LIN {X 0,Y 473.655,Z 542.16,A -85,B 0,C 180,E1 -7089.139,E2 -7089.139} C_VEL
LIN {X 0,Y 473.783,Z 539.256,A -85,B 0,C 180,E1 -7090.503,E2 -7090.503} C_VEL
LIN {X 0,Y 473.901,Z 535.976,A -85,B 0,C 180,E1 -7091.646,E2 -7091.646} C_VEL
LIN {X 0,Y 474,Z 531.987,A -85,B 0,C 180,E1 -7092.75,E2 -7092.75} C_VEL
LIN {X 0,Y 474.226,Z 525.864,A -85,B 0,C 180,E1 -7094.079,E2 -7094.079} C_VEL
LIN {X 0,Y 474.493,Z 519.562,A -85,B 0,C 180,E1 -7095.197,E2 -7095.197} C_VEL
LIN {X 0,Y 474.846,Z 511.99,A -85,B 0,C 180,E1 -7096.302,E2 -7096.302} C_VEL
LIN {X 0,Y 475.225,Z 503.778,A -85,B 0,C 180,E1 -7097.296,E2 -7097.296} C_VEL
LIN {X 0,Y 475.641,Z 495.123,A -85,B 0,C 180,E1 -7098.17,E2 -7098.17} C_VEL
LIN {X 0,Y 476.009,Z 486.024,A -85,B 0,C 180,E1 -7098.934,E2 -7098.934} C_VEL
LIN {X 0,Y 476.406,Z 476.552,A -85,B 0,C 180,E1 -7099.589,E2 -7099.589} C_VEL
LIN {X 0,Y 476.754,Z 465.648,A -85,B 0,C 180,E1 -7100.186,E2 -7100.186} C_VEL
LIN {X 0,Y 477.105,Z 454.466,A -85,B 0,C 180,E1 -7100.648,E2 -7100.648} C_VEL
LIN {X 0,Y 477.363,Z 443.291,A -85,B 0,C 180,E1 -7100.975,E2 -7100.975} C_VEL
LIN {X 0,Y 477.534,Z 425.281,A -85,B 0,C 180,E1 -7101.291,E2 -7101.291} C_VEL
LIN {X 0,Y 478.031,Z 348.456,A -85,B 0,C 180,E1 -7102.453,E2 -7102.453} C_VEL
LIN {X 0,Y 475.663,Z 335.476,A -85,B 0,C 180,E1 -7102.743,E2 -7102.743} C_VEL
LIN {X 0,Y 475.427,Z 333.673,A -85,B 0,C 180,E1 -7102.844,E2 -7102.844} C_VEL
LIN {X 0,Y 476.024,Z 317.906,A -85,B 0,C 180,E1 -7105.979,E2 -7105.979} C_VEL
LIN {X 0,Y 476.244,Z 312.656,A -85,B 0,C 180,E1 -7107.039,E2 -7107.039} C_VEL
LIN {X 0,Y 474.843,Z 303.952,A -85,B 0,C 180,E1 -7108.94,E2 -7108.94} C_VEL
LIN {X 0,Y 474.859,Z 303.836,A -85,B 0,C 180,E1 -7110.848,E2 -7110.848} C_VEL
LIN {X 0,Y 474.895,Z 303.831,A -85,B 0,C 180,E1 -7112.545,E2 -7112.545} C_VEL
LIN {X 0,Y 474.772,Z 303.839,A -85,B 0,C 180,E1 -7115.948,E2 -7115.948} C_VEL
LIN {X 0,Y 474.714,Z 303.846,A -85,B 0,C 180,E1 -7118.514,E2 -7118.514} C_VEL
LIN {X 0,Y 474.706,Z 303.85,A -85,B 0,C 180,E1 -7121.962,E2 -7121.962} C_VEL
LIN {X 0,Y 474.702,Z 303.851,A -85,B 0,C 180,E1 -7125.456,E2 -7125.456} C_VEL
LIN {X 0,Y 474.667,Z 303.85,A -85,B 0,C 180,E1 -7129.01,E2 -7129.01} C_VEL
LIN {X 0,Y 474.59,Z 303.863,A -85,B 0,C 180,E1 -7131.729,E2 -7131.729} C_VEL
LIN {X 0,Y 474.656,Z 303.858,A -85,B 0,C 180,E1 -7134.493,E2 -7134.493} C_VEL
LIN {X 0,Y 474.683,Z 303.85,A -85,B 0,C 180,E1 -7137.334,E2 -7137.334} C_VEL
LIN {X 0,Y 474.607,Z 303.859,A -85,B 0,C 180,E1 -7140.23,E2 -7140.23} C_VEL
LIN {X 0,Y 474.645,Z 303.861,A -85,B 0,C 180,E1 -7143.22,E2 -7143.22} C_VEL
LIN {X 0,Y 474.586,Z 303.864,A -85,B 0,C 180,E1 -7146.324,E2 -7146.324} C_VEL
LIN {X 0,Y 474.629,Z 303.861,A -85,B 0,C 180,E1 -7149.648,E2 -7149.648} C_VEL
LIN {X 0,Y 474.607,Z 303.857,A -85,B 0,C 180,E1 -7152.935,E2 -7152.935} C_VEL
LIN {X 0,Y 474.605,Z 303.861,A -85,B 0,C 180,E1 -7155.894,E2 -7155.894} C_VEL
LIN {X 0,Y 474.624,Z 303.854,A -85,B 0,C 180,E1 -7159.042,E2 -7159.042} C_VEL
LIN {X 0,Y 474.611,Z 303.854,A -85,B 0,C 180,E1 -7161.704,E2 -7161.704} C_VEL
LIN {X 0,Y 474.624,Z 303.858,A -85,B 0,C 180,E1 -7164.726,E2 -7164.726} C_VEL
LIN {X 0,Y 474.637,Z 303.856,A -85,B 0,C 180,E1 -7167.788,E2 -7167.788} C_VEL
LIN {X 0,Y 474.608,Z 303.845,A -85,B 0,C 180,E1 -7170.889,E2 -7170.889} C_VEL
LIN {X 0,Y 474.616,Z 303.856,A -85,B 0,C 180,E1 -7173.626,E2 -7173.626} C_VEL
LIN {X 0,Y 474.637,Z 303.86,A -85,B 0,C 180,E1 -7176.642,E2 -7176.642} C_VEL
LIN {X 0,Y 474.655,Z 303.849,A -85,B 0,C 180,E1 -7180.089,E2 -7180.089} C_VEL
LIN {X 0,Y 474.637,Z 303.847,A -85,B 0,C 180,E1 -7182.774,E2 -7182.774} C_VEL
LIN {X 0,Y 474.643,Z 303.859,A -85,B 0,C 180,E1 -7185.421,E2 -7185.421} C_VEL
LIN {X 0,Y 474.706,Z 303.848,A -85,B 0,C 180,E1 -7188.037,E2 -7188.037} C_VEL
LIN {X 0,Y 474.698,Z 303.85,A -85,B 0,C 180,E1 -7191.486,E2 -7191.486} C_VEL
LIN {X 0,Y 474.742,Z 303.836,A -85,B 0,C 180,E1 -7194.052,E2 -7194.052} C_VEL
LIN {X 0,Y 474.876,Z 303.824,A -85,B 0,C 180,E1 -7197.455,E2 -7197.455} C_VEL
LIN {X 0,Y 474.884,Z 303.828,A -85,B 0,C 180,E1 -7200,E2 -7200} C_VEL
LIN {X 0,Y 474.874,Z 303.828,A -85,B 0,C 180,E1 -7202.544,E2 -7202.544} C_VEL
LIN {X 0,Y 474.76,Z 303.83,A -85,B 0,C 180,E1 -7205.948,E2 -7205.948} C_VEL
LIN {X 0,Y 474.703,Z 303.847,A -85,B 0,C 180,E1 -7208.514,E2 -7208.514} C_VEL
LIN {X 0,Y 474.705,Z 303.847,A -85,B 0,C 180,E1 -7211.962,E2 -7211.962} C_VEL
LIN {X 0,Y 474.681,Z 303.845,A -85,B 0,C 180,E1 -7215.456,E2 -7215.456} C_VEL
LIN {X 0,Y 474.66,Z 303.853,A -85,B 0,C 180,E1 -7219.01,E2 -7219.01} C_VEL
LIN {X 0,Y 474.588,Z 303.863,A -85,B 0,C 180,E1 -7221.729,E2 -7221.729} C_VEL
LIN {X 0,Y 474.625,Z 303.857,A -85,B 0,C 180,E1 -7224.494,E2 -7224.494} C_VEL
LIN {X 0,Y 474.598,Z 303.863,A -85,B 0,C 180,E1 -7227.326,E2 -7227.326} C_VEL
LIN {X 0,Y 474.594,Z 303.858,A -85,B 0,C 180,E1 -7230.231,E2 -7230.231} C_VEL
LIN {X 0,Y 474.614,Z 303.864,A -85,B 0,C 180,E1 -7233.222,E2 -7233.222} C_VEL
LIN {X 0,Y 474.58,Z 303.861,A -85,B 0,C 180,E1 -7236.324,E2 -7236.324} C_VEL
LIN {X 0,Y 474.6,Z 303.866,A -85,B 0,C 180,E1 -7239.643,E2 -7239.643} C_VEL
LIN {X 0,Y 474.574,Z 303.868,A -85,B 0,C 180,E1 -7242.23,E2 -7242.23} C_VEL
LIN {X 0,Y 474.611,Z 303.859,A -85,B 0,C 180,E1 -7245.298,E2 -7245.298} C_VEL
LIN {X 0,Y 474.589,Z 303.866,A -85,B 0,C 180,E1 -7248.211,E2 -7248.211} C_VEL
LIN {X 0,Y 474.6,Z 303.862,A -85,B 0,C 180,E1 -7251.541,E2 -7251.541} C_VEL
LIN {X 0,Y 474.617,Z 303.862,A -85,B 0,C 180,E1 -7254.725,E2 -7254.725} C_VEL
LIN {X 0,Y 474.625,Z 303.864,A -85,B 0,C 180,E1 -7257.787,E2 -7257.787} C_VEL
LIN {X 0,Y 474.604,Z 303.864,A -85,B 0,C 180,E1 -7260.888,E2 -7260.888} C_VEL
LIN {X 0,Y 474.588,Z 303.868,A -85,B 0,C 180,E1 -7263.624,E2 -7263.624} C_VEL
LIN {X 0,Y 474.659,Z 304.014,A -85,B 0,C 180,E1 -7265.274,E2 -7265.274} C_VEL
LIN {X 0,Y 476.452,Z 313.581,A -85,B 0,C 180,E1 -7267.219,E2 -7267.219} C_VEL
LIN {X 0,Y 476.572,Z 317.444,A -85,B 0,C 180,E1 -7267.956,E2 -7267.956} C_VEL
LIN {X 0,Y 475.739,Z 335.291,A -85,B 0,C 180,E1 -7271.258,E2 -7271.258} C_VEL
LIN {X 0,Y 475.396,Z 346.264,A -85,B 0,C 180,E1 -7273.226,E2 -7273.226} C_VEL
LIN {X 0,Y 476.707,Z 354.719,A -85,B 0,C 180,E1 -7273.437,E2 -7273.437} C_VEL
LIN {X 0,Y 478.041,Z 363.134,A -85,B 0,C 180,E1 -7273.613,E2 -7273.613} C_VEL
LIN {X 0,Y 477.426,Z 452.372,A -85,B 0,C 180,E1 -7274.99,E2 -7274.99} C_VEL
LIN {X 0,Y 477.205,Z 462.229,A -85,B 0,C 180,E1 -7275.228,E2 -7275.228} C_VEL
LIN {X 0,Y 476.875,Z 472.814,A -85,B 0,C 180,E1 -7275.599,E2 -7275.599} C_VEL
LIN {X 0,Y 476.578,Z 482.083,A -85,B 0,C 180,E1 -7276.026,E2 -7276.026} C_VEL
LIN {X 0,Y 476.14,Z 493.305,A -85,B 0,C 180,E1 -7276.698,E2 -7276.698} C_VEL
LIN {X 0,Y 475.741,Z 502.94,A -85,B 0,C 180,E1 -7277.417,E2 -7277.417} C_VEL
LIN {X 0,Y 475.317,Z 512.31,A -85,B 0,C 180,E1 -7278.27,E2 -7278.27} C_VEL
LIN {X 0,Y 474.979,Z 520.193,A -85,B 0,C 180,E1 -7279.126,E2 -7279.126} C_VEL
LIN {X 0,Y 474.598,Z 528.371,A -85,B 0,C 180,E1 -7280.195,E2 -7280.195} C_VEL
LIN {X 0,Y 474.314,Z 535.182,A -85,B 0,C 180,E1 -7281.264,E2 -7281.264} C_VEL
LIN {X 0,Y 474.069,Z 540.876,A -85,B 0,C 180,E1 -7282.332,E2 -7282.332} C_VEL
LIN {X 0,Y 473.929,Z 545.951,A -85,B 0,C 180,E1 -7283.49,E2 -7283.49} C_VEL
LIN {X 0,Y 473.834,Z 550.733,A -85,B 0,C 180,E1 -7284.894,E2 -7284.894} C_VEL
LIN {X 0,Y 473.733,Z 553.044,A -85,B 0,C 180,E1 -7285.746,E2 -7285.746} C_VEL
LIN {X 0,Y 473.717,Z 556.305,A -85,B 0,C 180,E1 -7287.449,E2 -7287.449} C_VEL
LIN {X 0,Y 473.681,Z 557.843,A -85,B 0,C 180,E1 -7289.15,E2 -7289.15} C_VEL
LIN {X 0,Y 473.664,Z 558.137,A -85,B 0,C 180,E1 -7290,E2 -7290} C_VEL
LIN {X 0,Y 473.687,Z 557.271,A -85,B 0,C 180,E1 -7291.7,E2 -7291.7} C_VEL
LIN {X 0,Y 473.717,Z 556.304,A -85,B 0,C 180,E1 -7292.551,E2 -7292.551} C_VEL
LIN {X 0,Y 473.733,Z 553.044,A -85,B 0,C 180,E1 -7294.254,E2 -7294.254} C_VEL
LIN {X 0,Y 473.868,Z 549.438,A -85,B 0,C 180,E1 -7295.532,E2 -7295.532} C_VEL
LIN {X 0,Y 473.972,Z 544.709,A -85,B 0,C 180,E1 -7296.813,E2 -7296.813} C_VEL
LIN {X 0,Y 474.17,Z 538.712,A -85,B 0,C 180,E1 -7298.094,E2 -7298.094} C_VEL
LIN {X 0,Y 474.4,Z 532.643,A -85,B 0,C 180,E1 -7299.164,E2 -7299.164} C_VEL
LIN {X 0,Y 474.715,Z 525.324,A -85,B 0,C 180,E1 -7300.233,E2 -7300.233} C_VEL
LIN {X 0,Y 475.171,Z 516.421,A -85,B 0,C 180,E1 -7301.302,E2 -7301.302} C_VEL
LIN {X 0,Y 475.602,Z 507.884,A -85,B 0,C 180,E1 -7302.155,E2 -7302.155} C_VEL
LIN {X 0,Y 475.929,Z 498.455,A -85,B 0,C 180,E1 -7302.939,E2 -7302.939} C_VEL
LIN {X 0,Y 476.278,Z 489.644,A -85,B 0,C 180,E1 -7303.547,E2 -7303.547} C_VEL
LIN {X 0,Y 476.732,Z 477.751,A -85,B 0,C 180,E1 -7304.187,E2 -7304.187} C_VEL
LIN {X 0,Y 477.051,Z 467.383,A -85,B 0,C 180,E1 -7304.613,E2 -7304.613} C_VEL
LIN {X 0,Y 477.397,Z 456.571,A -85,B 0,C 180,E1 -7304.929,E2 -7304.929} C_VEL
LIN {X 0,Y 477.55,Z 438.378,A -85,B 0,C 180,E1 -7305.252,E2 -7305.252} C_VEL
LIN {X 0,Y 477.994,Z 362.184,A -85,B 0,C 180,E1 -7306.417,E2 -7306.417} C_VEL
LIN {X 0,Y 475.357,Z 346.208,A -85,B 0,C 180,E1 -7306.791,E2 -7306.791} C_VEL
LIN {X 0,Y 475.635,Z 337.488,A -85,B 0,C 180,E1 -7308.3,E2 -7308.3} C_VEL
LIN {X 0,Y 476.378,Z 319.034,A -85,B 0,C 180,E1 -7311.653,E2 -7311.653} C_VEL
LIN {X 0,Y 476.369,Z 312.947,A -85,B 0,C 180,E1 -7312.785,E2 -7312.785} C_VEL
LIN {X 0,Y 474.654,Z 303.952,A -85,B 0,C 180,E1 -7314.61,E2 -7314.61} C_VEL
LIN {X 0,Y 474.634,Z 303.862,A -85,B 0,C 180,E1 -7317.324,E2 -7317.324} C_VEL
LIN {X 0,Y 474.599,Z 303.869,A -85,B 0,C 180,E1 -7320.231,E2 -7320.231} C_VEL
LIN {X 0,Y 474.622,Z 303.86,A -85,B 0,C 180,E1 -7323.222,E2 -7323.222} C_VEL
LIN {X 0,Y 474.586,Z 303.869,A -85,B 0,C 180,E1 -7326.324,E2 -7326.324} C_VEL
LIN {X 0,Y 474.611,Z 303.857,A -85,B 0,C 180,E1 -7329.646,E2 -7329.646} C_VEL
LIN {X 0,Y 474.598,Z 303.863,A -85,B 0,C 180,E1 -7332.234,E2 -7332.234} C_VEL
LIN {X 0,Y 474.62,Z 303.867,A -85,B 0,C 180,E1 -7335.297,E2 -7335.297} C_VEL
LIN {X 0,Y 474.619,Z 303.858,A -85,B 0,C 180,E1 -7338.215,E2 -7338.215} C_VEL
LIN {X 0,Y 474.611,Z 303.866,A -85,B 0,C 180,E1 -7341.543,E2 -7341.543} C_VEL
LIN {X 0,Y 474.628,Z 303.856,A -85,B 0,C 180,E1 -7344.726,E2 -7344.726} C_VEL
LIN {X 0,Y 474.635,Z 303.86,A -85,B 0,C 180,E1 -7347.788,E2 -7347.788} C_VEL
LIN {X 0,Y 474.624,Z 303.861,A -85,B 0,C 180,E1 -7350.885,E2 -7350.885} C_VEL
LIN {X 0,Y 474.66,Z 303.853,A -85,B 0,C 180,E1 -7353.629,E2 -7353.629} C_VEL
LIN {X 0,Y 474.635,Z 303.862,A -85,B 0,C 180,E1 -7356.642,E2 -7356.642} C_VEL
LIN {X 0,Y 474.658,Z 303.853,A -85,B 0,C 180,E1 -7360.09,E2 -7360.09} C_VEL
LIN {X 0,Y 474.652,Z 303.854,A -85,B 0,C 180,E1 -7362.775,E2 -7362.775} C_VEL
LIN {X 0,Y 474.654,Z 303.86,A -85,B 0,C 180,E1 -7365.421,E2 -7365.421} C_VEL
LIN {X 0,Y 474.706,Z 303.853,A -85,B 0,C 180,E1 -7368.038,E2 -7368.038} C_VEL
LIN {X 0,Y 474.73,Z 303.843,A -85,B 0,C 180,E1 -7371.487,E2 -7371.487} C_VEL
LIN {X 0,Y 474.781,Z 303.847,A -85,B 0,C 180,E1 -7374.053,E2 -7374.053} C_VEL
LIN {X 0,Y 474.896,Z 303.824,A -85,B 0,C 180,E1 -7377.456,E2 -7377.456} C_VEL
LIN {X 0,Y 474.914,Z 303.822,A -85,B 0,C 180,E1 -7380,E2 -7380} C_VEL
LIN {X 0,Y 474.896,Z 303.83,A -85,B 0,C 180,E1 -7382.545,E2 -7382.545} C_VEL
LIN {X 0,Y 474.783,Z 303.838,A -85,B 0,C 180,E1 -7385.948,E2 -7385.948} C_VEL
LIN {X 0,Y 474.73,Z 303.845,A -85,B 0,C 180,E1 -7388.514,E2 -7388.514} C_VEL
LIN {X 0,Y 474.706,Z 303.848,A -85,B 0,C 180,E1 -7391.963,E2 -7391.963} C_VEL
LIN {X 0,Y 474.702,Z 303.855,A -85,B 0,C 180,E1 -7395.456,E2 -7395.456} C_VEL
LIN {X 0,Y 474.667,Z 303.852,A -85,B 0,C 180,E1 -7399.01,E2 -7399.01} C_VEL
LIN {X 0,Y 474.59,Z 303.867,A -85,B 0,C 180,E1 -7401.729,E2 -7401.729} C_VEL
LIN {X 0,Y 474.642,Z 303.863,A -85,B 0,C 180,E1 -7404.494,E2 -7404.494} C_VEL
LIN {X 0,Y 474.656,Z 303.849,A -85,B 0,C 180,E1 -7407.328,E2 -7407.328} C_VEL
LIN {X 0,Y 474.606,Z 303.865,A -85,B 0,C 180,E1 -7410.81,E2 -7410.81} C_VEL
LIN {X 0,Y 474.626,Z 303.862,A -85,B 0,C 180,E1 -7413.222,E2 -7413.222} C_VEL
LIN {X 0,Y 474.589,Z 303.863,A -85,B 0,C 180,E1 -7416.324,E2 -7416.324} C_VEL
LIN {X 0,Y 474.628,Z 303.865,A -85,B 0,C 180,E1 -7419.648,E2 -7419.648} C_VEL
LIN {X 0,Y 474.635,Z 303.864,A -85,B 0,C 180,E1 -7422.932,E2 -7422.932} C_VEL
LIN {X 0,Y 474.659,Z 304.019,A -85,B 0,C 180,E1 -7423.755,E2 -7423.755} C_VEL
LIN {X 0,Y 475.868,Z 310.991,A -85,B 0,C 180,E1 -7425.146,E2 -7425.146} C_VEL
LIN {X 0,Y 475.559,Z 326.316,A -85,B 0,C 180,E1 -7427.972,E2 -7427.972} C_VEL
LIN {X 0,Y 475.397,Z 333.585,A -85,B 0,C 180,E1 -7429.262,E2 -7429.262} C_VEL
LIN {X 0,Y 478.15,Z 348.867,A -85,B 0,C 180,E1 -7429.624,E2 -7429.624} C_VEL
LIN {X 0,Y 477.411,Z 440.006,A -85,B 0,C 180,E1 -7431.037,E2 -7431.037} C_VEL
LIN {X 0,Y 477.184,Z 449.685,A -85,B 0,C 180,E1 -7431.277,E2 -7431.277} C_VEL
LIN {X 0,Y 477.012,Z 458.923,A -85,B 0,C 180,E1 -7431.598,E2 -7431.598} C_VEL
LIN {X 0,Y 476.643,Z 470.39,A -85,B 0,C 180,E1 -7432.139,E2 -7432.139} C_VEL
LIN {X 0,Y 476.508,Z 473.811,A -85,B 0,C 180,E1 -7432.334,E2 -7432.334} C_VEL
LIN {X 0,Y 475.642,Z 479.172,A -85,B 0,C 180,E1 -7432.636,E2 -7432.636} C_VEL
LIN {X 0,Y 472.465,Z 487.502,A -85,B 0,C 180,E1 -7433.15,E2 -7433.15} C_VEL
LIN {X 0,Y 469.282,Z 495.478,A -85,B 0,C 180,E1 -7433.757,E2 -7433.757} C_VEL
LIN {X 0,Y 468.416,Z 500.019,A -85,B 0,C 180,E1 -7434.2,E2 -7434.2} C_VEL
LIN {X 0,Y 468.094,Z 506.843,A -85,B 0,C 180,E1 -7434.95,E2 -7434.95} C_VEL
LIN {X 0,Y 467.706,Z 514.606,A -85,B 0,C 180,E1 -7435.967,E2 -7435.967} C_VEL
LIN {X 0,Y 467.348,Z 522.436,A -85,B 0,C 180,E1 -7437.223,E2 -7437.223} C_VEL
LIN {X 0,Y 467.109,Z 527.684,A -85,B 0,C 180,E1 -7438.224,E2 -7438.224} C_VEL
LIN {X 0,Y 466.952,Z 532.064,A -85,B 0,C 180,E1 -7439.221,E2 -7439.221} C_VEL
LIN {X 0,Y 466.75,Z 537.603,A -85,B 0,C 180,E1 -7440.847,E2 -7440.847} C_VEL
LIN {X 0,Y 466.651,Z 540.911,A -85,B 0,C 180,E1 -7442.168,E2 -7442.168} C_VEL
LIN {X 0,Y 466.561,Z 542.715,A -85,B 0,C 180,E1 -7443.134,E2 -7443.134} C_VEL
LIN {X 0,Y 466.466,Z 544.498,A -85,B 0,C 180,E1 -7444.688,E2 -7444.688} C_VEL
LIN {X 0,Y 466.46,Z 544.981,A -85,B 0,C 180,E1 -7445.996,E2 -7445.996} C_VEL
LIN {X 0,Y 466.474,Z 544,A -85,B 0,C 180,E1 -7447.873,E2 -7447.873} C_VEL
LIN {X 0,Y 466.548,Z 542.49,A -85,B 0,C 180,E1 -7449.06,E2 -7449.06} C_VEL
LIN {X 0,Y 466.657,Z 540.335,A -85,B 0,C 180,E1 -7450.193,E2 -7450.193} C_VEL
LIN {X 0,Y 466.818,Z 536.626,A -85,B 0,C 180,E1 -7451.569,E2 -7451.569} C_VEL
LIN {X 0,Y 467.011,Z 530.719,A -85,B 0,C 180,E1 -7453.161,E2 -7453.161} C_VEL
LIN {X 0,Y 467.252,Z 524.78,A -85,B 0,C 180,E1 -7454.417,E2 -7454.417} C_VEL
LIN {X 0,Y 467.492,Z 519.119,A -85,B 0,C 180,E1 -7455.415,E2 -7455.415} C_VEL
LIN {X 0,Y 467.858,Z 511.447,A -85,B 0,C 180,E1 -7456.536,E2 -7456.536} C_VEL
LIN {X 0,Y 468.244,Z 503.727,A -85,B 0,C 180,E1 -7457.479,E2 -7457.479} C_VEL
LIN {X 0,Y 468.713,Z 494.292,A -85,B 0,C 180,E1 -7458.431,E2 -7458.431} C_VEL
LIN {X 0,Y 469.134,Z 484.967,A -85,B 0,C 180,E1 -7459.207,E2 -7459.207} C_VEL
LIN {X 0,Y 469.537,Z 475.223,A -85,B 0,C 180,E1 -7459.871,E2 -7459.871} C_VEL
LIN {X 0,Y 469.891,Z 465.105,A -85,B 0,C 180,E1 -7460.422,E2 -7460.422} C_VEL
LIN {X 0,Y 470.226,Z 454.023,A -85,B 0,C 180,E1 -7460.88,E2 -7460.88} C_VEL
LIN {X 0,Y 470.517,Z 443.081,A -85,B 0,C 180,E1 -7461.199,E2 -7461.199} C_VEL
LIN {X 0,Y 470.709,Z 424.841,A -85,B 0,C 180,E1 -7461.521,E2 -7461.521} C_VEL
LIN {X 0,Y 471.238,Z 349.532,A -85,B 0,C 180,E1 -7462.677,E2 -7462.677} C_VEL
LIN {X 0,Y 468.66,Z 335.347,A -85,B 0,C 180,E1 -7463.002,E2 -7463.002} C_VEL
LIN {X 0,Y 468.457,Z 333.704,A -85,B 0,C 180,E1 -7463.107,E2 -7463.107} C_VEL
LIN {X 0,Y 469.279,Z 315.538,A -85,B 0,C 180,E1 -7466.781,E2 -7466.781} C_VEL
LIN {X 0,Y 468.819,Z 310.492,A -85,B 0,C 180,E1 -7467.852,E2 -7467.852} C_VEL
LIN {X 0,Y 467.806,Z 304.81,A -85,B 0,C 180,E1 -7469.139,E2 -7469.139} C_VEL
LIN {X 0,Y 467.811,Z 304.714,A -85,B 0,C 180,E1 -7470.861,E2 -7470.861} C_VEL
LIN {X 0,Y 467.861,Z 304.707,A -85,B 0,C 180,E1 -7472.583,E2 -7472.583} C_VEL
LIN {X 0,Y 467.736,Z 304.715,A -85,B 0,C 180,E1 -7476.038,E2 -7476.038} C_VEL
LIN {X 0,Y 467.672,Z 304.724,A -85,B 0,C 180,E1 -7478.643,E2 -7478.643} C_VEL
LIN {X 0,Y 467.658,Z 304.726,A -85,B 0,C 180,E1 -7482.146,E2 -7482.146} C_VEL
LIN {X 0,Y 467.641,Z 304.733,A -85,B 0,C 180,E1 -7485.695,E2 -7485.695} C_VEL
LIN {X 0,Y 467.619,Z 304.729,A -85,B 0,C 180,E1 -7488.765,E2 -7488.765} C_VEL
LIN {X 0,Y 467.582,Z 304.736,A -85,B 0,C 180,E1 -7491.268,E2 -7491.268} C_VEL
LIN {X 0,Y 467.572,Z 304.734,A -85,B 0,C 180,E1 -7493.943,E2 -7493.943} C_VEL
LIN {X 0,Y 467.618,Z 304.738,A -85,B 0,C 180,E1 -7496.8,E2 -7496.8} C_VEL
LIN {X 0,Y 467.556,Z 304.739,A -85,B 0,C 180,E1 -7499.738,E2 -7499.738} C_VEL
LIN {X 0,Y 467.585,Z 304.735,A -85,B 0,C 180,E1 -7502.758,E2 -7502.758} C_VEL
LIN {X 0,Y 467.552,Z 304.745,A -85,B 0,C 180,E1 -7505.89,E2 -7505.89} C_VEL
LIN {X 0,Y 467.583,Z 304.735,A -85,B 0,C 180,E1 -7509.145,E2 -7509.145} C_VEL
LIN {X 0,Y 467.588,Z 304.735,A -85,B 0,C 180,E1 -7512.567,E2 -7512.567} C_VEL
LIN {X 0,Y 467.567,Z 304.739,A -85,B 0,C 180,E1 -7515.053,E2 -7515.053} C_VEL
LIN {X 0,Y 467.575,Z 304.74,A -85,B 0,C 180,E1 -7518.597,E2 -7518.597} C_VEL
LIN {X 0,Y 467.566,Z 304.73,A -85,B 0,C 180,E1 -7521.955,E2 -7521.955} C_VEL
LIN {X 0,Y 467.561,Z 304.744,A -85,B 0,C 180,E1 -7525.167,E2 -7525.167} C_VEL
LIN {X 0,Y 467.585,Z 304.729,A -85,B 0,C 180,E1 -7528.26,E2 -7528.26} C_VEL
LIN {X 0,Y 467.557,Z 304.724,A -85,B 0,C 180,E1 -7531.249,E2 -7531.249} C_VEL
LIN {X 0,Y 467.585,Z 304.74,A -85,B 0,C 180,E1 -7534.158,E2 -7534.158} C_VEL
LIN {X 0,Y 467.578,Z 304.736,A -85,B 0,C 180,E1 -7536.996,E2 -7536.996} C_VEL
LIN {X 0,Y 467.624,Z 304.723,A -85,B 0,C 180,E1 -7539.777,E2 -7539.777} C_VEL
LIN {X 0,Y 467.597,Z 304.719,A -85,B 0,C 180,E1 -7542.506,E2 -7542.506} C_VEL
LIN {X 0,Y 467.603,Z 304.737,A -85,B 0,C 180,E1 -7545.196,E2 -7545.196} C_VEL
LIN {X 0,Y 467.658,Z 304.727,A -85,B 0,C 180,E1 -7547.854,E2 -7547.854} C_VEL
LIN {X 0,Y 467.658,Z 304.726,A -85,B 0,C 180,E1 -7551.357,E2 -7551.357} C_VEL
LIN {X 0,Y 467.706,Z 304.711,A -85,B 0,C 180,E1 -7553.962,E2 -7553.962} C_VEL
LIN {X 0,Y 467.817,Z 304.703,A -85,B 0,C 180,E1 -7557.417,E2 -7557.417} C_VEL
LIN {X 0,Y 467.854,Z 304.704,A -85,B 0,C 180,E1 -7560,E2 -7560} C_VEL
LIN {X 0,Y 467.815,Z 304.706,A -85,B 0,C 180,E1 -7562.583,E2 -7562.583} C_VEL
LIN {X 0,Y 467.724,Z 304.707,A -85,B 0,C 180,E1 -7566.037,E2 -7566.037} C_VEL
LIN {X 0,Y 467.662,Z 304.725,A -85,B 0,C 180,E1 -7568.643,E2 -7568.643} C_VEL
LIN {X 0,Y 467.657,Z 304.724,A -85,B 0,C 180,E1 -7572.145,E2 -7572.145} C_VEL
LIN {X 0,Y 467.606,Z 304.727,A -85,B 0,C 180,E1 -7575.696,E2 -7575.696} C_VEL
LIN {X 0,Y 467.62,Z 304.731,A -85,B 0,C 180,E1 -7579.308,E2 -7579.308} C_VEL
LIN {X 0,Y 467.535,Z 304.745,A -85,B 0,C 180,E1 -7582.074,E2 -7582.074} C_VEL
LIN {X 0,Y 467.555,Z 304.74,A -85,B 0,C 180,E1 -7584.89,E2 -7584.89} C_VEL
LIN {X 0,Y 467.545,Z 304.74,A -85,B 0,C 180,E1 -7587.774,E2 -7587.774} C_VEL
LIN {X 0,Y 467.547,Z 304.741,A -85,B 0,C 180,E1 -7591.04,E2 -7591.04} C_VEL
LIN {X 0,Y 467.575,Z 304.737,A -85,B 0,C 180,E1 -7594.239,E2 -7594.239} C_VEL
LIN {X 0,Y 467.536,Z 304.74,A -85,B 0,C 180,E1 -7597.184,E2 -7597.184} C_VEL
LIN {X 0,Y 467.555,Z 304.743,A -85,B 0,C 180,E1 -7600.267,E2 -7600.267} C_VEL
LIN {X 0,Y 467.516,Z 304.745,A -85,B 0,C 180,E1 -7602.568,E2 -7602.568} C_VEL
LIN {X 0,Y 467.56,Z 304.739,A -85,B 0,C 180,E1 -7605.052,E2 -7605.052} C_VEL
LIN {X 0,Y 467.558,Z 304.745,A -85,B 0,C 180,E1 -7608.726,E2 -7608.726} C_VEL
LIN {X 0,Y 467.553,Z 304.739,A -85,B 0,C 180,E1 -7611.954,E2 -7611.954} C_VEL
LIN {X 0,Y 467.554,Z 304.747,A -85,B 0,C 180,E1 -7615.166,E2 -7615.166} C_VEL
LIN {X 0,Y 467.576,Z 304.738,A -85,B 0,C 180,E1 -7618.259,E2 -7618.259} C_VEL
LIN {X 0,Y 467.552,Z 304.745,A -85,B 0,C 180,E1 -7621.249,E2 -7621.249} C_VEL
LIN {X 0,Y 467.565,Z 304.745,A -85,B 0,C 180,E1 -7624.157,E2 -7624.157} C_VEL
LIN {X 0,Y 467.617,Z 304.876,A -85,B 0,C 180,E1 -7625.061,E2 -7625.061} C_VEL
LIN {X 0,Y 469.618,Z 315.892,A -85,B 0,C 180,E1 -7627.334,E2 -7627.334} C_VEL
LIN {X 0,Y 469.158,Z 326.746,A -85,B 0,C 180,E1 -7629.388,E2 -7629.388} C_VEL
LIN {X 0,Y 468.442,Z 343.624,A -85,B 0,C 180,E1 -7632.539,E2 -7632.539} C_VEL
LIN {X 0,Y 468.408,Z 346.284,A -85,B 0,C 180,E1 -7632.98,E2 -7632.98} C_VEL
LIN {X 0,Y 471.217,Z 363.856,A -85,B 0,C 180,E1 -7633.385,E2 -7633.385} C_VEL
LIN {X 0,Y 470.588,Z 452.076,A -85,B 0,C 180,E1 -7634.766,E2 -7634.766} C_VEL
LIN {X 0,Y 470.35,Z 462.005,A -85,B 0,C 180,E1 -7635.008,E2 -7635.008} C_VEL
LIN {X 0,Y 470.004,Z 472.627,A -85,B 0,C 180,E1 -7635.384,E2 -7635.384} C_VEL
LIN {X 0,Y 469.697,Z 481.92,A -85,B 0,C 180,E1 -7635.817,E2 -7635.817} C_VEL
LIN {X 0,Y 469.224,Z 493.159,A -85,B 0,C 180,E1 -7636.499,E2 -7636.499} C_VEL
LIN {X 0,Y 468.853,Z 502.059,A -85,B 0,C 180,E1 -7637.162,E2 -7637.162} C_VEL
LIN {X 0,Y 468.357,Z 512.184,A -85,B 0,C 180,E1 -7638.093,E2 -7638.093} C_VEL
LIN {X 0,Y 467.956,Z 520.072,A -85,B 0,C 180,E1 -7638.96,E2 -7638.96} C_VEL
LIN {X 0,Y 467.59,Z 528.255,A -85,B 0,C 180,E1 -7640.046,E2 -7640.046} C_VEL
LIN {X 0,Y 467.279,Z 535.069,A -85,B 0,C 180,E1 -7641.132,E2 -7641.132} C_VEL
LIN {X 0,Y 467.022,Z 540.766,A -85,B 0,C 180,E1 -7642.216,E2 -7642.216} C_VEL
LIN {X 0,Y 466.844,Z 546.236,A -85,B 0,C 180,E1 -7643.502,E2 -7643.502} C_VEL
LIN {X 0,Y 466.767,Z 550.629,A -85,B 0,C 180,E1 -7644.817,E2 -7644.817} C_VEL
LIN {X 0,Y 466.645,Z 552.94,A -85,B 0,C 180,E1 -7645.681,E2 -7645.681} C_VEL
LIN {X 0,Y 466.638,Z 556.205,A -85,B 0,C 180,E1 -7647.41,E2 -7647.41} C_VEL
LIN {X 0,Y 466.583,Z 557.743,A -85,B 0,C 180,E1 -7649.137,E2 -7649.137} C_VEL
LIN {X 0,Y 466.593,Z 558.038,A -85,B 0,C 180,E1 -7650,E2 -7650} C_VEL
LIN {X 0,Y 466.597,Z 557.173,A -85,B 0,C 180,E1 -7651.726,E2 -7651.726} C_VEL
LIN {X 0,Y 466.638,Z 556.205,A -85,B 0,C 180,E1 -7652.59,E2 -7652.59} C_VEL
LIN {X 0,Y 466.645,Z 552.945,A -85,B 0,C 180,E1 -7654.319,E2 -7654.319} C_VEL
LIN {X 0,Y 466.782,Z 549.338,A -85,B 0,C 180,E1 -7655.616,E2 -7655.616} C_VEL
LIN {X 0,Y 466.907,Z 544.609,A -85,B 0,C 180,E1 -7656.916,E2 -7656.916} C_VEL
LIN {X 0,Y 467.112,Z 538.61,A -85,B 0,C 180,E1 -7658.218,E2 -7658.218} C_VEL
LIN {X 0,Y 467.367,Z 532.54,A -85,B 0,C 180,E1 -7659.303,E2 -7659.303} C_VEL
LIN {X 0,Y 467.693,Z 525.222,A -85,B 0,C 180,E1 -7660.389,E2 -7660.389} C_VEL
LIN {X 0,Y 468.198,Z 516.324,A -85,B 0,C 180,E1 -7661.472,E2 -7661.472} C_VEL
LIN {X 0,Y 468.64,Z 508.001,A -85,B 0,C 180,E1 -7662.32,E2 -7662.32} C_VEL
LIN {X 0,Y 469.04,Z 497.629,A -85,B 0,C 180,E1 -7663.187,E2 -7663.187} C_VEL
LIN {X 0,Y 469.426,Z 487.695,A -85,B 0,C 180,E1 -7663.86,E2 -7663.86} C_VEL
LIN {X 0,Y 469.852,Z 477.695,A -85,B 0,C 180,E1 -7664.399,E2 -7664.399} C_VEL
LIN {X 0,Y 470.204,Z 466.518,A -85,B 0,C 180,E1 -7664.858,E2 -7664.858} C_VEL
LIN {X 0,Y 470.529,Z 456.577,A -85,B 0,C 180,E1 -7665.152,E2 -7665.152} C_VEL
LIN {X 0,Y 470.715,Z 438.43,A -85,B 0,C 180,E1 -7665.479,E2 -7665.479} C_VEL
LIN {X 0,Y 471.125,Z 362.415,A -85,B 0,C 180,E1 -7666.661,E2 -7666.661} C_VEL
LIN {X 0,Y 468.401,Z 346.178,A -85,B 0,C 180,E1 -7667.046,E2 -7667.046} C_VEL
LIN {X 0,Y 468.418,Z 343.519,A -85,B 0,C 180,E1 -7667.462,E2 -7667.462} C_VEL
LIN {X 0,Y 469.04,Z 328.808,A -85,B 0,C 180,E1 -7670.159,E2 -7670.159} C_VEL
LIN {X 0,Y 469.551,Z 315.308,A -85,B 0,C 180,E1 -7672.669,E2 -7672.669} C_VEL
LIN {X 0,Y 467.603,Z 304.959,A -85,B 0,C 180,E1 -7674.769,E2 -7674.769} C_VEL
LIN {X 0,Y 467.576,Z 304.744,A -85,B 0,C 180,E1 -7677.772,E2 -7677.772} C_VEL
LIN {X 0,Y 467.564,Z 304.74,A -85,B 0,C 180,E1 -7681.045,E2 -7681.045} C_VEL
LIN {X 0,Y 467.575,Z 304.74,A -85,B 0,C 180,E1 -7684.24,E2 -7684.24} C_VEL
LIN {X 0,Y 467.546,Z 304.744,A -85,B 0,C 180,E1 -7687.186,E2 -7687.186} C_VEL
LIN {X 0,Y 467.57,Z 304.735,A -85,B 0,C 180,E1 -7690.265,E2 -7690.265} C_VEL
LIN {X 0,Y 467.549,Z 304.743,A -85,B 0,C 180,E1 -7693.745,E2 -7693.745} C_VEL
LIN {X 0,Y 467.555,Z 304.739,A -85,B 0,C 180,E1 -7696.256,E2 -7696.256} C_VEL
LIN {X 0,Y 467.577,Z 304.734,A -85,B 0,C 180,E1 -7698.723,E2 -7698.723} C_VEL
LIN {X 0,Y 467.565,Z 304.745,A -85,B 0,C 180,E1 -7701.956,E2 -7701.956} C_VEL
LIN {X 0,Y 467.567,Z 304.735,A -85,B 0,C 180,E1 -7705.168,E2 -7705.168} C_VEL
LIN {X 0,Y 467.582,Z 304.74,A -85,B 0,C 180,E1 -7708.26,E2 -7708.26} C_VEL
LIN {X 0,Y 467.577,Z 304.736,A -85,B 0,C 180,E1 -7711.251,E2 -7711.251} C_VEL
LIN {X 0,Y 467.616,Z 304.732,A -85,B 0,C 180,E1 -7713.2,E2 -7713.2} C_VEL
LIN {X 0,Y 467.592,Z 304.737,A -85,B 0,C 180,E1 -7716.469,E2 -7716.469} C_VEL
LIN {X 0,Y 467.625,Z 304.731,A -85,B 0,C 180,E1 -7719.778,E2 -7719.778} C_VEL
LIN {X 0,Y 467.61,Z 304.73,A -85,B 0,C 180,E1 -7722.507,E2 -7722.507} C_VEL
LIN {X 0,Y 467.611,Z 304.737,A -85,B 0,C 180,E1 -7725.197,E2 -7725.197} C_VEL
LIN {X 0,Y 467.657,Z 304.733,A -85,B 0,C 180,E1 -7727.855,E2 -7727.855} C_VEL
LIN {X 0,Y 467.684,Z 304.72,A -85,B 0,C 180,E1 -7731.358,E2 -7731.358} C_VEL
LIN {X 0,Y 467.746,Z 304.722,A -85,B 0,C 180,E1 -7733.963,E2 -7733.963} C_VEL
LIN {X 0,Y 467.861,Z 304.7,A -85,B 0,C 180,E1 -7737.417,E2 -7737.417} C_VEL
LIN {X 0,Y 467.885,Z 304.698,A -85,B 0,C 180,E1 -7740,E2 -7740} C_VEL
LIN {X 0,Y 467.861,Z 304.707,A -85,B 0,C 180,E1 -7742.583,E2 -7742.583} C_VEL
LIN {X 0,Y 467.748,Z 304.714,A -85,B 0,C 180,E1 -7746.038,E2 -7746.038} C_VEL
LIN {X 0,Y 467.684,Z 304.724,A -85,B 0,C 180,E1 -7748.643,E2 -7748.643} C_VEL
LIN {X 0,Y 467.658,Z 304.724,A -85,B 0,C 180,E1 -7752.146,E2 -7752.146} C_VEL
LIN {X 0,Y 467.641,Z 304.734,A -85,B 0,C 180,E1 -7755.695,E2 -7755.695} C_VEL
LIN {X 0,Y 467.619,Z 304.73,A -85,B 0,C 180,E1 -7758.765,E2 -7758.765} C_VEL
LIN {X 0,Y 467.582,Z 304.736,A -85,B 0,C 180,E1 -7761.268,E2 -7761.268} C_VEL
LIN {X 0,Y 467.564,Z 304.743,A -85,B 0,C 180,E1 -7763.944,E2 -7763.944} C_VEL
LIN {X 0,Y 467.577,Z 304.736,A -85,B 0,C 180,E1 -7766.803,E2 -7766.803} C_VEL
LIN {X 0,Y 467.549,Z 304.741,A -85,B 0,C 180,E1 -7769.739,E2 -7769.739} C_VEL
LIN {X 0,Y 467.58,Z 304.743,A -85,B 0,C 180,E1 -7772.759,E2 -7772.759} C_VEL
LIN {X 0,Y 467.554,Z 304.74,A -85,B 0,C 180,E1 -7775.89,E2 -7775.89} C_VEL
LIN {X 0,Y 467.583,Z 304.742,A -85,B 0,C 180,E1 -7779.145,E2 -7779.145} C_VEL
LIN {X 0,Y 467.588,Z 304.742,A -85,B 0,C 180,E1 -7782.567,E2 -7782.567} C_VEL
LIN {X 0,Y 467.62,Z 304.979,A -85,B 0,C 180,E1 -7783.588,E2 -7783.588} C_VEL
LIN {X 0,Y 468.882,Z 311.995,A -85,B 0,C 180,E1 -7785.005,E2 -7785.005} C_VEL
LIN {X 0,Y 468.639,Z 325.644,A -85,B 0,C 180,E1 -7787.558,E2 -7787.558} C_VEL
LIN {X 0,Y 468.455,Z 333.676,A -85,B 0,C 180,E1 -7788.999,E2 -7788.999} C_VEL
LIN {X 0,Y 471.352,Z 349.794,A -85,B 0,C 180,E1 -7789.39,E2 -7789.39} C_VEL
LIN {X 0,Y 470.58,Z 439.751,A -85,B 0,C 180,E1 -7790.804,E2 -7790.804} C_VEL
LIN {X 0,Y 470.35,Z 449.748,A -85,B 0,C 180,E1 -7791.053,E2 -7791.053} C_VEL
LIN {X 0,Y 470.1,Z 460.538,A -85,B 0,C 180,E1 -7791.448,E2 -7791.448} C_VEL
LIN {X 0,Y 469.735,Z 471.011,A -85,B 0,C 180,E1 -7791.959,E2 -7791.959} C_VEL
LIN {X 0,Y 469.382,Z 480.178,A -85,B 0,C 180,E1 -7792.52,E2 -7792.52} C_VEL
LIN {X 0,Y 468.898,Z 490.393,A -85,B 0,C 180,E1 -7793.298,E2 -7793.298} C_VEL
LIN {X 0,Y 468.421,Z 499.903,A -85,B 0,C 180,E1 -7794.187,E2 -7794.187} C_VEL
LIN {X 0,Y 468.416,Z 500.019,A -85,B 0,C 180,E1 -7794.2,E2 -7794.2} C_VEL
LIN {X 0,Y 467.559,Z 504.594,A -85,B 0,C 180,E1 -7794.669,E2 -7794.669} C_VEL
LIN {X 0,Y 464.366,Z 511.43,A -85,B 0,C 180,E1 -7795.448,E2 -7795.448} C_VEL
LIN {X 0,Y 461.181,Z 517.821,A -85,B 0,C 180,E1 -7796.297,E2 -7796.297} C_VEL
LIN {X 0,Y 460.328,Z 521.388,A -85,B 0,C 180,E1 -7796.871,E2 -7796.871} C_VEL
LIN {X 0,Y 460.025,Z 528.182,A -85,B 0,C 180,E1 -7798.192,E2 -7798.192} C_VEL
LIN {X 0,Y 459.883,Z 532.784,A -85,B 0,C 180,E1 -7799.273,E2 -7799.273} C_VEL
LIN {X 0,Y 459.7,Z 537.56,A -85,B 0,C 180,E1 -7800.71,E2 -7800.71} C_VEL
LIN {X 0,Y 459.592,Z 540.159,A -85,B 0,C 180,E1 -7801.703,E2 -7801.703} C_VEL
LIN {X 0,Y 459.479,Z 542.077,A -85,B 0,C 180,E1 -7802.686,E2 -7802.686} C_VEL
LIN {X 0,Y 459.372,Z 544.469,A -85,B 0,C 180,E1 -7804.509,E2 -7804.509} C_VEL
LIN {X 0,Y 459.361,Z 544.95,A -85,B 0,C 180,E1 -7805.601,E2 -7805.601} C_VEL
LIN {X 0,Y 459.369,Z 544.516,A -85,B 0,C 180,E1 -7807.513,E2 -7807.513} C_VEL
LIN {X 0,Y 459.456,Z 542.922,A -85,B 0,C 180,E1 -7808.92,E2 -7808.92} C_VEL
LIN {X 0,Y 459.589,Z 540.223,A -85,B 0,C 180,E1 -7810.341,E2 -7810.341} C_VEL
LIN {X 0,Y 459.741,Z 536.181,A -85,B 0,C 180,E1 -7811.811,E2 -7811.811} C_VEL
LIN {X 0,Y 459.926,Z 531.443,A -85,B 0,C 180,E1 -7813.122,E2 -7813.122} C_VEL
LIN {X 0,Y 460.12,Z 526.624,A -85,B 0,C 180,E1 -7814.213,E2 -7814.213} C_VEL
LIN {X 0,Y 460.432,Z 520.129,A -85,B 0,C 180,E1 -7815.413,E2 -7815.413} C_VEL
LIN {X 0,Y 460.814,Z 512.63,A -85,B 0,C 180,E1 -7816.551,E2 -7816.551} C_VEL
LIN {X 0,Y 461.283,Z 503.493,A -85,B 0,C 180,E1 -7817.684,E2 -7817.684} C_VEL
LIN {X 0,Y 461.745,Z 494.687,A -85,B 0,C 180,E1 -7818.588,E2 -7818.588} C_VEL
LIN {X 0,Y 462.184,Z 485.428,A -85,B 0,C 180,E1 -7819.375,E2 -7819.375} C_VEL
LIN {X 0,Y 462.609,Z 475.768,A -85,B 0,C 180,E1 -7820.049,E2 -7820.049} C_VEL
LIN {X 0,Y 462.999,Z 465.313,A -85,B 0,C 180,E1 -7820.629,E2 -7820.629} C_VEL
LIN {X 0,Y 463.362,Z 454.292,A -85,B 0,C 180,E1 -7821.093,E2 -7821.093} C_VEL
LIN {X 0,Y 463.671,Z 443.309,A -85,B 0,C 180,E1 -7821.419,E2 -7821.419} C_VEL
LIN {X 0,Y 463.851,Z 426.569,A -85,B 0,C 180,E1 -7821.724,E2 -7821.724} C_VEL
LIN {X 0,Y 464.435,Z 350.426,A -85,B 0,C 180,E1 -7822.91,E2 -7822.91} C_VEL
LIN {X 0,Y 461.604,Z 334.944,A -85,B 0,C 180,E1 -7823.279,E2 -7823.279} C_VEL
LIN {X 0,Y 461.507,Z 333.681,A -85,B 0,C 180,E1 -7823.387,E2 -7823.387} C_VEL
LIN {X 0,Y 462.333,Z 316.343,A -85,B 0,C 180,E1 -7826.95,E2 -7826.95} C_VEL
LIN {X 0,Y 461.587,Z 310.34,A -85,B 0,C 180,E1 -7828.255,E2 -7828.255} C_VEL
LIN {X 0,Y 460.808,Z 305.661,A -85,B 0,C 180,E1 -7829.345,E2 -7829.345} C_VEL
LIN {X 0,Y 460.825,Z 305.584,A -85,B 0,C 180,E1 -7832.622,E2 -7832.622} C_VEL
LIN {X 0,Y 460.702,Z 305.592,A -85,B 0,C 180,E1 -7836.13,E2 -7836.13} C_VEL
LIN {X 0,Y 460.622,Z 305.603,A -85,B 0,C 180,E1 -7838.776,E2 -7838.776} C_VEL
LIN {X 0,Y 460.615,Z 305.602,A -85,B 0,C 180,E1 -7842.445,E2 -7842.445} C_VEL
LIN {X 0,Y 460.602,Z 305.611,A -85,B 0,C 180,E1 -7845.998,E2 -7845.998} C_VEL
LIN {X 0,Y 460.573,Z 305.606,A -85,B 0,C 180,E1 -7848.902,E2 -7848.902} C_VEL
LIN {X 0,Y 460.518,Z 305.616,A -85,B 0,C 180,E1 -7851.486,E2 -7851.486} C_VEL
LIN {X 0,Y 460.54,Z 305.614,A -85,B 0,C 180,E1 -7854.333,E2 -7854.333} C_VEL
LIN {X 0,Y 460.574,Z 305.608,A -85,B 0,C 180,E1 -7857.244,E2 -7857.244} C_VEL
LIN {X 0,Y 460.512,Z 305.615,A -85,B 0,C 180,E1 -7860.24,E2 -7860.24} C_VEL
LIN {X 0,Y 460.531,Z 305.617,A -85,B 0,C 180,E1 -7863.325,E2 -7863.325} C_VEL
LIN {X 0,Y 460.474,Z 305.62,A -85,B 0,C 180,E1 -7866.53,E2 -7866.53} C_VEL
LIN {X 0,Y 460.559,Z 305.616,A -85,B 0,C 180,E1 -7869.86,E2 -7869.86} C_VEL
LIN {X 0,Y 460.513,Z 305.613,A -85,B 0,C 180,E1 -7872.9,E2 -7872.9} C_VEL
LIN {X 0,Y 460.507,Z 305.617,A -85,B 0,C 180,E1 -7875.831,E2 -7875.831} C_VEL
LIN {X 0,Y 460.529,Z 305.61,A -85,B 0,C 180,E1 -7878.988,E2 -7878.988} C_VEL
LIN {X 0,Y 460.519,Z 305.613,A -85,B 0,C 180,E1 -7881.266,E2 -7881.266} C_VEL
LIN {X 0,Y 460.51,Z 305.616,A -85,B 0,C 180,E1 -7884.554,E2 -7884.554} C_VEL
LIN {X 0,Y 460.532,Z 305.614,A -85,B 0,C 180,E1 -7887.716,E2 -7887.716} C_VEL
LIN {X 0,Y 460.528,Z 305.598,A -85,B 0,C 180,E1 -7890.768,E2 -7890.768} C_VEL
LIN {X 0,Y 460.533,Z 305.612,A -85,B 0,C 180,E1 -7893.733,E2 -7893.733} C_VEL
LIN {X 0,Y 460.546,Z 305.616,A -85,B 0,C 180,E1 -7896.624,E2 -7896.624} C_VEL
LIN {X 0,Y 460.553,Z 305.604,A -85,B 0,C 180,E1 -7899.453,E2 -7899.453} C_VEL
LIN {X 0,Y 460.549,Z 305.594,A -85,B 0,C 180,E1 -7902.23,E2 -7902.23} C_VEL
LIN {X 0,Y 460.564,Z 305.609,A -85,B 0,C 180,E1 -7904.965,E2 -7904.965} C_VEL
LIN {X 0,Y 460.61,Z 305.603,A -85,B 0,C 180,E1 -7908.559,E2 -7908.559} C_VEL
LIN {X 0,Y 460.611,Z 305.602,A -85,B 0,C 180,E1 -7911.223,E2 -7911.223} C_VEL
LIN {X 0,Y 460.672,Z 305.586,A -85,B 0,C 180,E1 -7913.869,E2 -7913.869} C_VEL
LIN {X 0,Y 460.761,Z 305.581,A -85,B 0,C 180,E1 -7917.377,E2 -7917.377} C_VEL
LIN {X 0,Y 460.823,Z 305.58,A -85,B 0,C 180,E1 -7920,E2 -7920} C_VEL
LIN {X 0,Y 460.759,Z 305.584,A -85,B 0,C 180,E1 -7922.623,E2 -7922.623} C_VEL
LIN {X 0,Y 460.69,Z 305.583,A -85,B 0,C 180,E1 -7926.13,E2 -7926.13} C_VEL
LIN {X 0,Y 460.613,Z 305.604,A -85,B 0,C 180,E1 -7928.776,E2 -7928.776} C_VEL
LIN {X 0,Y 460.598,Z 305.602,A -85,B 0,C 180,E1 -7932.435,E2 -7932.435} C_VEL
LIN {X 0,Y 460.558,Z 305.608,A -85,B 0,C 180,E1 -7935.978,E2 -7935.978} C_VEL
LIN {X 0,Y 460.566,Z 305.611,A -85,B 0,C 180,E1 -7939.615,E2 -7939.615} C_VEL
LIN {X 0,Y 460.511,Z 305.616,A -85,B 0,C 180,E1 -7942.428,E2 -7942.428} C_VEL
LIN {X 0,Y 460.532,Z 305.61,A -85,B 0,C 180,E1 -7945.792,E2 -7945.792} C_VEL
LIN {X 0,Y 460.52,Z 305.617,A -85,B 0,C 180,E1 -7949.232,E2 -7949.232} C_VEL
LIN {X 0,Y 460.524,Z 305.61,A -85,B 0,C 180,E1 -7952.285,E2 -7952.285} C_VEL
LIN {X 0,Y 460.505,Z 305.625,A -85,B 0,C 180,E1 -7955.446,E2 -7955.446} C_VEL
LIN {X 0,Y 460.492,Z 305.617,A -85,B 0,C 180,E1 -7958.889,E2 -7958.889} C_VEL
LIN {X 0,Y 460.5,Z 305.62,A -85,B 0,C 180,E1 -7961.598,E2 -7961.598} C_VEL
LIN {X 0,Y 460.508,Z 305.622,A -85,B 0,C 180,E1 -7964.589,E2 -7964.589} C_VEL
LIN {X 0,Y 460.471,Z 305.622,A -85,B 0,C 180,E1 -7967.813,E2 -7967.813} C_VEL
LIN {X 0,Y 460.509,Z 305.618,A -85,B 0,C 180,E1 -7970.135,E2 -7970.135} C_VEL
LIN {X 0,Y 460.469,Z 305.626,A -85,B 0,C 180,E1 -7973.47,E2 -7973.47} C_VEL
LIN {X 0,Y 460.514,Z 305.613,A -85,B 0,C 180,E1 -7976.674,E2 -7976.674} C_VEL
LIN {X 0,Y 460.504,Z 305.624,A -85,B 0,C 180,E1 -7979.759,E2 -7979.759} C_VEL
LIN {X 0,Y 460.527,Z 305.618,A -85,B 0,C 180,E1 -7982.753,E2 -7982.753} C_VEL
LIN {X 0,Y 460.543,Z 305.71,A -85,B 0,C 180,E1 -7984.825,E2 -7984.825} C_VEL
LIN {X 0,Y 462.487,Z 315.77,A -85,B 0,C 180,E1 -7986.964,E2 -7986.964} C_VEL
LIN {X 0,Y 462.729,Z 319.405,A -85,B 0,C 180,E1 -7987.685,E2 -7987.685} C_VEL
LIN {X 0,Y 461.81,Z 336.773,A -85,B 0,C 180,E1 -7990.994,E2 -7990.994} C_VEL
LIN {X 0,Y 461.431,Z 346.124,A -85,B 0,C 180,E1 -7992.715,E2 -7992.715} C_VEL
LIN {X 0,Y 464.403,Z 364.317,A -85,B 0,C 180,E1 -7993.145,E2 -7993.145} C_VEL
LIN {X 0,Y 463.743,Z 451.703,A -85,B 0,C 180,E1 -7994.536,E2 -7994.536} C_VEL
LIN {X 0,Y 463.5,Z 461.729,A -85,B 0,C 180,E1 -7994.781,E2 -7994.781} C_VEL
LIN {X 0,Y 463.134,Z 472.398,A -85,B 0,C 180,E1 -7995.163,E2 -7995.163} C_VEL
LIN {X 0,Y 462.682,Z 483.591,A -85,B 0,C 180,E1 -7995.71,E2 -7995.71} C_VEL
LIN {X 0,Y 462.251,Z 494.031,A -85,B 0,C 180,E1 -7996.369,E2 -7996.369} C_VEL
LIN {X 0,Y 461.852,Z 502.676,A -85,B 0,C 180,E1 -7997.035,E2 -7997.035} C_VEL
LIN {X 0,Y 461.396,Z 512.033,A -85,B 0,C 180,E1 -7997.91,E2 -7997.91} C_VEL
LIN {X 0,Y 460.968,Z 519.933,A -85,B 0,C 180,E1 -7998.791,E2 -7998.791} C_VEL
LIN {X 0,Y 460.543,Z 528.126,A -85,B 0,C 180,E1 -7999.893,E2 -7999.893} C_VEL
LIN {X 0,Y 460.208,Z 534.948,A -85,B 0,C 180,E1 -8000.994,E2 -8000.994} C_VEL
LIN {X 0,Y 459.96,Z 540.652,A -85,B 0,C 180,E1 -8002.096,E2 -8002.096} C_VEL
LIN {X 0,Y 459.76,Z 546.515,A -85,B 0,C 180,E1 -8003.514,E2 -8003.514} C_VEL
LIN {X 0,Y 459.678,Z 550.524,A -85,B 0,C 180,E1 -8004.737,E2 -8004.737} C_VEL
LIN {X 0,Y 459.563,Z 552.836,A -85,B 0,C 180,E1 -8005.615,E2 -8005.615} C_VEL
LIN {X 0,Y 459.561,Z 556.104,A -85,B 0,C 180,E1 -8007.37,E2 -8007.37} C_VEL
LIN {X 0,Y 459.488,Z 557.643,A -85,B 0,C 180,E1 -8009.124,E2 -8009.124} C_VEL
LIN {X 0,Y 459.495,Z 557.939,A -85,B 0,C 180,E1 -8010,E2 -8010} C_VEL
LIN {X 0,Y 459.509,Z 557.074,A -85,B 0,C 180,E1 -8011.753,E2 -8011.753} C_VEL
LIN {X 0,Y 459.561,Z 556.106,A -85,B 0,C 180,E1 -8012.629,E2 -8012.629} C_VEL
LIN {X 0,Y 459.563,Z 552.848,A -85,B 0,C 180,E1 -8014.385,E2 -8014.385} C_VEL
LIN {X 0,Y 459.698,Z 549.242,A -85,B 0,C 180,E1 -8015.703,E2 -8015.703} C_VEL
LIN {X 0,Y 459.842,Z 544.515,A -85,B 0,C 180,E1 -8017.023,E2 -8017.023} C_VEL
LIN {X 0,Y 460.071,Z 538.52,A -85,B 0,C 180,E1 -8018.344,E2 -8018.344} C_VEL
LIN {X 0,Y 460.337,Z 532.454,A -85,B 0,C 180,E1 -8019.446,E2 -8019.446} C_VEL
LIN {X 0,Y 460.68,Z 525.139,A -85,B 0,C 180,E1 -8020.548,E2 -8020.548} C_VEL
LIN {X 0,Y 461.217,Z 516.244,A -85,B 0,C 180,E1 -8021.648,E2 -8021.648} C_VEL
LIN {X 0,Y 461.675,Z 508.135,A -85,B 0,C 180,E1 -8022.489,E2 -8022.489} C_VEL
LIN {X 0,Y 462.111,Z 497.557,A -85,B 0,C 180,E1 -8023.388,E2 -8023.388} C_VEL
LIN {X 0,Y 462.528,Z 487.63,A -85,B 0,C 180,E1 -8024.07,E2 -8024.07} C_VEL
LIN {X 0,Y 462.992,Z 477.642,A -85,B 0,C 180,E1 -8024.617,E2 -8024.617} C_VEL
LIN {X 0,Y 463.329,Z 467.313,A -85,B 0,C 180,E1 -8025.056,E2 -8025.056} C_VEL
LIN {X 0,Y 463.685,Z 456.583,A -85,B 0,C 180,E1 -8025.381,E2 -8025.381} C_VEL
LIN {X 0,Y 463.888,Z 438.482,A -85,B 0,C 180,E1 -8025.712,E2 -8025.712} C_VEL
LIN {X 0,Y 464.362,Z 363.486,A -85,B 0,C 180,E1 -8026.896,E2 -8026.896} C_VEL
LIN {X 0,Y 461.422,Z 345.961,A -85,B 0,C 180,E1 -8027.324,E2 -8027.324} C_VEL
LIN {X 0,Y 461.533,Z 342.197,A -85,B 0,C 180,E1 -8027.96,E2 -8027.96} C_VEL
LIN {X 0,Y 462.189,Z 326.257,A -85,B 0,C 180,E1 -8030.937,E2 -8030.937} C_VEL
LIN {X 0,Y 462.643,Z 317.671,A -85,B 0,C 180,E1 -8032.555,E2 -8032.555} C_VEL
LIN {X 0,Y 461.239,Z 309.064,A -85,B 0,C 180,E1 -8034.293,E2 -8034.293} C_VEL
LIN {X 0,Y 460.545,Z 305.676,A -85,B 0,C 180,E1 -8035.054,E2 -8035.054} C_VEL
LIN {X 0,Y 460.522,Z 305.622,A -85,B 0,C 180,E1 -8038.235,E2 -8038.235} C_VEL
LIN {X 0,Y 460.517,Z 305.618,A -85,B 0,C 180,E1 -8041.283,E2 -8041.283} C_VEL
LIN {X 0,Y 460.521,Z 305.621,A -85,B 0,C 180,E1 -8044.504,E2 -8044.504} C_VEL
LIN {X 0,Y 460.499,Z 305.619,A -85,B 0,C 180,E1 -8047.623,E2 -8047.623} C_VEL
LIN {X 0,Y 460.534,Z 305.611,A -85,B 0,C 180,E1 -8050.269,E2 -8050.269} C_VEL
LIN {X 0,Y 460.508,Z 305.623,A -85,B 0,C 180,E1 -8053.374,E2 -8053.374} C_VEL
LIN {X 0,Y 460.498,Z 305.618,A -85,B 0,C 180,E1 -8056.625,E2 -8056.625} C_VEL
LIN {X 0,Y 460.538,Z 305.622,A -85,B 0,C 180,E1 -8059.731,E2 -8059.731} C_VEL
LIN {X 0,Y 460.499,Z 305.62,A -85,B 0,C 180,E1 -8062.524,E2 -8062.524} C_VEL
LIN {X 0,Y 460.547,Z 305.612,A -85,B 0,C 180,E1 -8065.624,E2 -8065.624} C_VEL
LIN {X 0,Y 460.537,Z 305.615,A -85,B 0,C 180,E1 -8068.745,E2 -8068.745} C_VEL
LIN {X 0,Y 460.588,Z 305.611,A -85,B 0,C 180,E1 -8072.252,E2 -8072.252} C_VEL
LIN {X 0,Y 460.558,Z 305.619,A -85,B 0,C 180,E1 -8074.706,E2 -8074.706} C_VEL
LIN {X 0,Y 460.511,Z 305.616,A -85,B 0,C 180,E1 -8077.572,E2 -8077.572} C_VEL
LIN {X 0,Y 460.57,Z 305.609,A -85,B 0,C 180,E1 -8080.385,E2 -8080.385} C_VEL
LIN {X 0,Y 460.566,Z 305.613,A -85,B 0,C 180,E1 -8083.147,E2 -8083.147} C_VEL
LIN {X 0,Y 460.559,Z 305.61,A -85,B 0,C 180,E1 -8085.868,E2 -8085.868} C_VEL
LIN {X 0,Y 460.613,Z 305.604,A -85,B 0,C 180,E1 -8088.56,E2 -8088.56} C_VEL
LIN {X 0,Y 460.697,Z 305.599,A -85,B 0,C 180,E1 -8092.109,E2 -8092.109} C_VEL
LIN {X 0,Y 460.7,Z 305.592,A -85,B 0,C 180,E1 -8094.749,E2 -8094.749} C_VEL
LIN {X 0,Y 460.826,Z 305.576,A -85,B 0,C 180,E1 -8097.378,E2 -8097.378} C_VEL
LIN {X 0,Y 460.856,Z 305.573,A -85,B 0,C 180,E1 -8100,E2 -8100} C_VEL
LIN {X 0,Y 460.826,Z 305.584,A -85,B 0,C 180,E1 -8102.623,E2 -8102.623} C_VEL
LIN {X 0,Y 460.714,Z 305.591,A -85,B 0,C 180,E1 -8106.13,E2 -8106.13} C_VEL
LIN {X 0,Y 460.631,Z 305.603,A -85,B 0,C 180,E1 -8108.776,E2 -8108.776} C_VEL
LIN {X 0,Y 460.615,Z 305.601,A -85,B 0,C 180,E1 -8112.445,E2 -8112.445} C_VEL
LIN {X 0,Y 460.602,Z 305.61,A -85,B 0,C 180,E1 -8115.998,E2 -8115.998} C_VEL
LIN {X 0,Y 460.573,Z 305.607,A -85,B 0,C 180,E1 -8118.902,E2 -8118.902} C_VEL
LIN {X 0,Y 460.517,Z 305.618,A -85,B 0,C 180,E1 -8121.486,E2 -8121.486} C_VEL
LIN {X 0,Y 460.532,Z 305.621,A -85,B 0,C 180,E1 -8124.333,E2 -8124.333} C_VEL
LIN {X 0,Y 460.566,Z 305.604,A -85,B 0,C 180,E1 -8127.742,E2 -8127.742} C_VEL
LIN {X 0,Y 460.522,Z 305.618,A -85,B 0,C 180,E1 -8131.283,E2 -8131.283} C_VEL
LIN {X 0,Y 460.524,Z 305.615,A -85,B 0,C 180,E1 -8134.504,E2 -8134.504} C_VEL
LIN {X 0,Y 460.502,Z 305.623,A -85,B 0,C 180,E1 -8137.623,E2 -8137.623} C_VEL
LIN {X 0,Y 460.543,Z 305.618,A -85,B 0,C 180,E1 -8140.269,E2 -8140.269} C_VEL
LIN {X 0,Y 460.588,Z 305.779,A -85,B 0,C 180,E1 -8143.365,E2 -8143.365} C_VEL
LIN {X 0,Y 461.976,Z 313.712,A -85,B 0,C 180,E1 -8144.995,E2 -8144.995} C_VEL
LIN {X 0,Y 461.642,Z 327.733,A -85,B 0,C 180,E1 -8147.65,E2 -8147.65} C_VEL
LIN {X 0,Y 461.519,Z 333.7,A -85,B 0,C 180,E1 -8148.722,E2 -8148.722} C_VEL
LIN {X 0,Y 463.236,Z 343.115,A -85,B 0,C 180,E1 -8148.975,E2 -8148.975} C_VEL
LIN {X 0,Y 464.565,Z 350.649,A -85,B 0,C 180,E1 -8149.149,E2 -8149.149} C_VEL
LIN {X 0,Y 463.745,Z 440.001,A -85,B 0,C 180,E1 -8150.575,E2 -8150.575} C_VEL
LIN {X 0,Y 463.507,Z 450.022,A -85,B 0,C 180,E1 -8150.83,E2 -8150.83} C_VEL
LIN {X 0,Y 463.287,Z 459.925,A -85,B 0,C 180,E1 -8151.193,E2 -8151.193} C_VEL
LIN {X 0,Y 462.902,Z 470.485,A -85,B 0,C 180,E1 -8151.706,E2 -8151.706} C_VEL
LIN {X 0,Y 462.44,Z 481.08,A -85,B 0,C 180,E1 -8152.37,E2 -8152.37} C_VEL
LIN {X 0,Y 461.983,Z 490.102,A -85,B 0,C 180,E1 -8153.066,E2 -8153.066} C_VEL
LIN {X 0,Y 461.517,Z 498.897,A -85,B 0,C 180,E1 -8153.884,E2 -8153.884} C_VEL
LIN {X 0,Y 461.077,Z 507.412,A -85,B 0,C 180,E1 -8154.838,E2 -8154.838} C_VEL
LIN {X 0,Y 460.656,Z 515.272,A -85,B 0,C 180,E1 -8155.897,E2 -8155.897} C_VEL
LIN {X 0,Y 460.328,Z 521.388,A -85,B 0,C 180,E1 -8156.871,E2 -8156.871} C_VEL
LIN {X 0,Y 459.498,Z 524.727,A -85,B 0,C 180,E1 -8157.471,E2 -8157.471} C_VEL
LIN {X 0,Y 457.775,Z 527.861,A -85,B 0,C 180,E1 -8158.07,E2 -8158.07} C_VEL
LIN {X 0,Y 453.862,Z 533.321,A -85,B 0,C 180,E1 -8159.312,E2 -8159.312} C_VEL
LIN {X 0,Y 452.752,Z 535.686,A -85,B 0,C 180,E1 -8159.981,E2 -8159.981} C_VEL
LIN {X 0,Y 452.65,Z 536.44,A -85,B 0,C 180,E1 -8160.211,E2 -8160.211} C_VEL
LIN {X 0,Y 452.494,Z 540.488,A -85,B 0,C 180,E1 -8161.724,E2 -8161.724} C_VEL
LIN {X 0,Y 452.33,Z 543.201,A -85,B 0,C 180,E1 -8163.219,E2 -8163.219} C_VEL
LIN {X 0,Y 452.275,Z 544.403,A -85,B 0,C 180,E1 -8164.326,E2 -8164.326} C_VEL
LIN {X 0,Y 452.256,Z 545.16,A -85,B 0,C 180,E1 -8166.169,E2 -8166.169} C_VEL
LIN {X 0,Y 452.257,Z 544.808,A -85,B 0,C 180,E1 -8167.139,E2 -8167.139} C_VEL
LIN {X 0,Y 452.379,Z 542.839,A -85,B 0,C 180,E1 -8169.064,E2 -8169.064} C_VEL
LIN {X 0,Y 452.53,Z 540.088,A -85,B 0,C 180,E1 -8170.494,E2 -8170.494} C_VEL
LIN {X 0,Y 452.658,Z 536.234,A -85,B 0,C 180,E1 -8171.909,E2 -8171.909} C_VEL
LIN {X 0,Y 452.889,Z 531.16,A -85,B 0,C 180,E1 -8173.317,E2 -8173.317} C_VEL
LIN {X 0,Y 453.088,Z 526.274,A -85,B 0,C 180,E1 -8174.422,E2 -8174.422} C_VEL
LIN {X 0,Y 453.427,Z 519.672,A -85,B 0,C 180,E1 -8175.641,E2 -8175.641} C_VEL
LIN {X 0,Y 453.821,Z 512.322,A -85,B 0,C 180,E1 -8176.762,E2 -8176.762} C_VEL
LIN {X 0,Y 454.293,Z 503.842,A -85,B 0,C 180,E1 -8177.832,E2 -8177.832} C_VEL
LIN {X 0,Y 454.778,Z 495.084,A -85,B 0,C 180,E1 -8178.749,E2 -8178.749} C_VEL
LIN {X 0,Y 455.264,Z 485.87,A -85,B 0,C 180,E1 -8179.55,E2 -8179.55} C_VEL
LIN {X 0,Y 455.709,Z 476.292,A -85,B 0,C 180,E1 -8180.233,E2 -8180.233} C_VEL
LIN {X 0,Y 456.106,Z 466.159,A -85,B 0,C 180,E1 -8180.813,E2 -8180.813} C_VEL
LIN {X 0,Y 456.501,Z 454.595,A -85,B 0,C 180,E1 -8181.311,E2 -8181.311} C_VEL
LIN {X 0,Y 456.84,Z 443.257,A -85,B 0,C 180,E1 -8181.652,E2 -8181.652} C_VEL
LIN {X 0,Y 457.014,Z 426.52,A -85,B 0,C 180,E1 -8181.961,E2 -8181.961} C_VEL
LIN {X 0,Y 457.539,Z 350.791,A -85,B 0,C 180,E1 -8183.163,E2 -8183.163} C_VEL
LIN {X 0,Y 454.618,Z 334.573,A -85,B 0,C 180,E1 -8183.565,E2 -8183.565} C_VEL
LIN {X 0,Y 454.574,Z 333.032,A -85,B 0,C 180,E1 -8183.787,E2 -8183.787} C_VEL
LIN {X 0,Y 455.364,Z 317.149,A -85,B 0,C 180,E1 -8187.125,E2 -8187.125} C_VEL
LIN {X 0,Y 454.356,Z 310.195,A -85,B 0,C 180,E1 -8188.671,E2 -8188.671} C_VEL
LIN {X 0,Y 453.793,Z 306.515,A -85,B 0,C 180,E1 -8189.556,E2 -8189.556} C_VEL
LIN {X 0,Y 453.766,Z 306.464,A -85,B 0,C 180,E1 -8192.663,E2 -8192.663} C_VEL
LIN {X 0,Y 453.669,Z 306.468,A -85,B 0,C 180,E1 -8196.226,E2 -8196.226} C_VEL
LIN {X 0,Y 453.588,Z 306.48,A -85,B 0,C 180,E1 -8198.914,E2 -8198.914} C_VEL
LIN {X 0,Y 453.565,Z 306.48,A -85,B 0,C 180,E1 -8202.529,E2 -8202.529} C_VEL
LIN {X 0,Y 453.547,Z 306.49,A -85,B 0,C 180,E1 -8206.196,E2 -8206.196} C_VEL
LIN {X 0,Y 453.522,Z 306.484,A -85,B 0,C 180,E1 -8209.041,E2 -8209.041} C_VEL
LIN {X 0,Y 453.478,Z 306.494,A -85,B 0,C 180,E1 -8211.836,E2 -8211.836} C_VEL
LIN {X 0,Y 453.509,Z 306.496,A -85,B 0,C 180,E1 -8214.735,E2 -8214.735} C_VEL
LIN {X 0,Y 453.534,Z 306.48,A -85,B 0,C 180,E1 -8217.96,E2 -8217.96} C_VEL
LIN {X 0,Y 453.468,Z 306.498,A -85,B 0,C 180,E1 -8221.525,E2 -8221.525} C_VEL
LIN {X 0,Y 453.488,Z 306.483,A -85,B 0,C 180,E1 -8224.777,E2 -8224.777} C_VEL
LIN {X 0,Y 453.465,Z 306.497,A -85,B 0,C 180,E1 -8228.312,E2 -8228.312} C_VEL
LIN {X 0,Y 453.496,Z 306.484,A -85,B 0,C 180,E1 -8230.609,E2 -8230.609} C_VEL
LIN {X 0,Y 453.454,Z 306.491,A -85,B 0,C 180,E1 -8233.244,E2 -8233.244} C_VEL
LIN {X 0,Y 453.462,Z 306.495,A -85,B 0,C 180,E1 -8235.778,E2 -8235.778} C_VEL
LIN {X 0,Y 453.495,Z 306.48,A -85,B 0,C 180,E1 -8239.409,E2 -8239.409} C_VEL
LIN {X 0,Y 453.454,Z 306.492,A -85,B 0,C 180,E1 -8242.81,E2 -8242.81} C_VEL
LIN {X 0,Y 453.47,Z 306.493,A -85,B 0,C 180,E1 -8246.087,E2 -8246.087} C_VEL
LIN {X 0,Y 453.477,Z 306.487,A -85,B 0,C 180,E1 -8249.24,E2 -8249.24} C_VEL
LIN {X 0,Y 453.509,Z 306.487,A -85,B 0,C 180,E1 -8252.296,E2 -8252.296} C_VEL
LIN {X 0,Y 453.497,Z 306.489,A -85,B 0,C 180,E1 -8255.264,E2 -8255.264} C_VEL
LIN {X 0,Y 453.483,Z 306.496,A -85,B 0,C 180,E1 -8258.415,E2 -8258.415} C_VEL
LIN {X 0,Y 453.525,Z 306.472,A -85,B 0,C 180,E1 -8261.009,E2 -8261.009} C_VEL
LIN {X 0,Y 453.572,Z 306.472,A -85,B 0,C 180,E1 -8263.88,E2 -8263.88} C_VEL
LIN {X 0,Y 453.566,Z 306.487,A -85,B 0,C 180,E1 -8267.471,E2 -8267.471} C_VEL
LIN {X 0,Y 453.578,Z 306.476,A -85,B 0,C 180,E1 -8271.086,E2 -8271.086} C_VEL
LIN {X 0,Y 453.639,Z 306.46,A -85,B 0,C 180,E1 -8273.774,E2 -8273.774} C_VEL
LIN {X 0,Y 453.708,Z 306.46,A -85,B 0,C 180,E1 -8277.336,E2 -8277.336} C_VEL
LIN {X 0,Y 453.793,Z 306.456,A -85,B 0,C 180,E1 -8280,E2 -8280} C_VEL
LIN {X 0,Y 453.705,Z 306.461,A -85,B 0,C 180,E1 -8282.663,E2 -8282.663} C_VEL
LIN {X 0,Y 453.657,Z 306.459,A -85,B 0,C 180,E1 -8286.225,E2 -8286.225} C_VEL
LIN {X 0,Y 453.58,Z 306.482,A -85,B 0,C 180,E1 -8288.913,E2 -8288.913} C_VEL
LIN {X 0,Y 453.566,Z 306.478,A -85,B 0,C 180,E1 -8292.529,E2 -8292.529} C_VEL
LIN {X 0,Y 453.498,Z 306.488,A -85,B 0,C 180,E1 -8296.197,E2 -8296.197} C_VEL
LIN {X 0,Y 453.518,Z 306.487,A -85,B 0,C 180,E1 -8299.039,E2 -8299.039} C_VEL
LIN {X 0,Y 453.477,Z 306.493,A -85,B 0,C 180,E1 -8301.836,E2 -8301.836} C_VEL
LIN {X 0,Y 453.486,Z 306.491,A -85,B 0,C 180,E1 -8304.736,E2 -8304.736} C_VEL
LIN {X 0,Y 453.462,Z 306.494,A -85,B 0,C 180,E1 -8307.942,E2 -8307.942} C_VEL
LIN {X 0,Y 453.456,Z 306.495,A -85,B 0,C 180,E1 -8310.761,E2 -8310.761} C_VEL
LIN {X 0,Y 453.466,Z 306.496,A -85,B 0,C 180,E1 -8313.913,E2 -8313.913} C_VEL
LIN {X 0,Y 453.445,Z 306.496,A -85,B 0,C 180,E1 -8317.19,E2 -8317.19} C_VEL
LIN {X 0,Y 453.469,Z 306.494,A -85,B 0,C 180,E1 -8320.611,E2 -8320.611} C_VEL
LIN {X 0,Y 453.478,Z 306.498,A -85,B 0,C 180,E1 -8324.528,E2 -8324.528} C_VEL
LIN {X 0,Y 453.44,Z 306.501,A -85,B 0,C 180,E1 -8328.205,E2 -8328.205} C_VEL
LIN {X 0,Y 453.443,Z 306.506,A -85,B 0,C 180,E1 -8330.801,E2 -8330.801} C_VEL
LIN {X 0,Y 453.448,Z 306.497,A -85,B 0,C 180,E1 -8333.916,E2 -8333.916} C_VEL
LIN {X 0,Y 453.473,Z 306.495,A -85,B 0,C 180,E1 -8337.15,E2 -8337.15} C_VEL
LIN {X 0,Y 453.464,Z 306.499,A -85,B 0,C 180,E1 -8340.267,E2 -8340.267} C_VEL
LIN {X 0,Y 453.46,Z 306.498,A -85,B 0,C 180,E1 -8343.291,E2 -8343.291} C_VEL
LIN {X 0,Y 453.528,Z 306.694,A -85,B 0,C 180,E1 -8344.654,E2 -8344.654} C_VEL
LIN {X 0,Y 455.658,Z 318.068,A -85,B 0,C 180,E1 -8347.079,E2 -8347.079} C_VEL
LIN {X 0,Y 455.558,Z 323.063,A -85,B 0,C 180,E1 -8348.062,E2 -8348.062} C_VEL
LIN {X 0,Y 454.711,Z 339.789,A -85,B 0,C 180,E1 -8351.294,E2 -8351.294} C_VEL
LIN {X 0,Y 454.476,Z 346.037,A -85,B 0,C 180,E1 -8352.451,E2 -8352.451} C_VEL
LIN {X 0,Y 457.62,Z 365.122,A -85,B 0,C 180,E1 -8352.908,E2 -8352.908} C_VEL
LIN {X 0,Y 456.865,Z 452.622,A -85,B 0,C 180,E1 -8354.326,E2 -8354.326} C_VEL
LIN {X 0,Y 456.619,Z 462.283,A -85,B 0,C 180,E1 -8354.575,E2 -8354.575} C_VEL
LIN {X 0,Y 456.278,Z 472.169,A -85,B 0,C 180,E1 -8354.934,E2 -8354.934} C_VEL
LIN {X 0,Y 455.79,Z 483.391,A -85,B 0,C 180,E1 -8355.489,E2 -8355.489} C_VEL
LIN {X 0,Y 455.344,Z 493.851,A -85,B 0,C 180,E1 -8356.159,E2 -8356.159} C_VEL
LIN {X 0,Y 454.854,Z 503.424,A -85,B 0,C 180,E1 -8356.916,E2 -8356.916} C_VEL
LIN {X 0,Y 454.429,Z 511.88,A -85,B 0,C 180,E1 -8357.722,E2 -8357.722} C_VEL
LIN {X 0,Y 453.992,Z 519.79,A -85,B 0,C 180,E1 -8358.616,E2 -8358.616} C_VEL
LIN {X 0,Y 453.52,Z 527.99,A -85,B 0,C 180,E1 -8359.734,E2 -8359.734} C_VEL
LIN {X 0,Y 453.15,Z 534.819,A -85,B 0,C 180,E1 -8360.853,E2 -8360.853} C_VEL
LIN {X 0,Y 452.899,Z 540.529,A -85,B 0,C 180,E1 -8361.972,E2 -8361.972} C_VEL
LIN {X 0,Y 452.717,Z 546.064,A -85,B 0,C 180,E1 -8363.314,E2 -8363.314} C_VEL
LIN {X 0,Y 452.593,Z 550.411,A -85,B 0,C 180,E1 -8364.654,E2 -8364.654} C_VEL
LIN {X 0,Y 452.486,Z 552.724,A -85,B 0,C 180,E1 -8365.546,E2 -8365.546} C_VEL
LIN {X 0,Y 452.485,Z 556,A -85,B 0,C 180,E1 -8367.329,E2 -8367.329} C_VEL
LIN {X 0,Y 452.397,Z 557.543,A -85,B 0,C 180,E1 -8369.11,E2 -8369.11} C_VEL
LIN {X 0,Y 452.401,Z 557.84,A -85,B 0,C 180,E1 -8370,E2 -8370} C_VEL
LIN {X 0,Y 452.426,Z 556.979,A -85,B 0,C 180,E1 -8371.78,E2 -8371.78} C_VEL
LIN {X 0,Y 452.485,Z 556.01,A -85,B 0,C 180,E1 -8372.671,E2 -8372.671} C_VEL
LIN {X 0,Y 452.486,Z 552.757,A -85,B 0,C 180,E1 -8374.454,E2 -8374.454} C_VEL
LIN {X 0,Y 452.599,Z 549.152,A -85,B 0,C 180,E1 -8375.793,E2 -8375.793} C_VEL
LIN {X 0,Y 452.756,Z 544.427,A -85,B 0,C 180,E1 -8377.133,E2 -8377.133} C_VEL
LIN {X 0,Y 453.013,Z 538.433,A -85,B 0,C 180,E1 -8378.475,E2 -8378.475} C_VEL
LIN {X 0,Y 453.297,Z 532.369,A -85,B 0,C 180,E1 -8379.594,E2 -8379.594} C_VEL
LIN {X 0,Y 453.674,Z 525.057,A -85,B 0,C 180,E1 -8380.713,E2 -8380.713} C_VEL
LIN {X 0,Y 454.237,Z 516.163,A -85,B 0,C 180,E1 -8381.83,E2 -8381.83} C_VEL
LIN {X 0,Y 454.71,Z 508.271,A -85,B 0,C 180,E1 -8382.664,E2 -8382.664} C_VEL
LIN {X 0,Y 455.155,Z 498.684,A -85,B 0,C 180,E1 -8383.506,E2 -8383.506} C_VEL
LIN {X 0,Y 455.568,Z 489.439,A -85,B 0,C 180,E1 -8384.176,E2 -8384.176} C_VEL
LIN {X 0,Y 456.13,Z 477.588,A -85,B 0,C 180,E1 -8384.842,E2 -8384.842} C_VEL
LIN {X 0,Y 456.53,Z 466.449,A -85,B 0,C 180,E1 -8385.314,E2 -8385.314} C_VEL
LIN {X 0,Y 456.835,Z 456.589,A -85,B 0,C 180,E1 -8385.618,E2 -8385.618} C_VEL
LIN {X 0,Y 457.072,Z 440.318,A -85,B 0,C 180,E1 -8385.924,E2 -8385.924} C_VEL
LIN {X 0,Y 457.559,Z 364.193,A -85,B 0,C 180,E1 -8387.145,E2 -8387.145} C_VEL
LIN {X 0,Y 454.459,Z 345.904,A -85,B 0,C 180,E1 -8387.598,E2 -8387.598} C_VEL
LIN {X 0,Y 454.589,Z 342.121,A -85,B 0,C 180,E1 -8388.244,E2 -8388.244} C_VEL
LIN {X 0,Y 455.333,Z 326.172,A -85,B 0,C 180,E1 -8391.267,E2 -8391.267} C_VEL
LIN {X 0,Y 455.702,Z 318.811,A -85,B 0,C 180,E1 -8392.678,E2 -8392.678} C_VEL
LIN {X 0,Y 453.991,Z 308.971,A -85,B 0,C 180,E1 -8394.707,E2 -8394.707} C_VEL
LIN {X 0,Y 453.508,Z 306.538,A -85,B 0,C 180,E1 -8395.286,E2 -8395.286} C_VEL
LIN {X 0,Y 453.489,Z 306.497,A -85,B 0,C 180,E1 -8398.713,E2 -8398.713} C_VEL
LIN {X 0,Y 453.46,Z 306.498,A -85,B 0,C 180,E1 -8401.8,E2 -8401.8} C_VEL
LIN {X 0,Y 453.474,Z 306.499,A -85,B 0,C 180,E1 -8404.99,E2 -8404.99} C_VEL
LIN {X 0,Y 453.46,Z 306.498,A -85,B 0,C 180,E1 -8408.312,E2 -8408.312} C_VEL
LIN {X 0,Y 453.491,Z 306.49,A -85,B 0,C 180,E1 -8410.609,E2 -8410.609} C_VEL
LIN {X 0,Y 453.461,Z 306.496,A -85,B 0,C 180,E1 -8414.222,E2 -8414.222} C_VEL
LIN {X 0,Y 453.462,Z 306.498,A -85,B 0,C 180,E1 -8417.005,E2 -8417.005} C_VEL
LIN {X 0,Y 453.493,Z 306.495,A -85,B 0,C 180,E1 -8419.409,E2 -8419.409} C_VEL
LIN {X 0,Y 453.449,Z 306.501,A -85,B 0,C 180,E1 -8422.227,E2 -8422.227} C_VEL
LIN {X 0,Y 453.488,Z 306.488,A -85,B 0,C 180,E1 -8425.223,E2 -8425.223} C_VEL
LIN {X 0,Y 453.466,Z 306.497,A -85,B 0,C 180,E1 -8428.475,E2 -8428.475} C_VEL
LIN {X 0,Y 453.537,Z 306.487,A -85,B 0,C 180,E1 -8432.039,E2 -8432.039} C_VEL
LIN {X 0,Y 453.512,Z 306.49,A -85,B 0,C 180,E1 -8435.266,E2 -8435.266} C_VEL
LIN {X 0,Y 453.48,Z 306.492,A -85,B 0,C 180,E1 -8438.415,E2 -8438.415} C_VEL
LIN {X 0,Y 453.523,Z 306.491,A -85,B 0,C 180,E1 -8441.009,E2 -8441.009} C_VEL
LIN {X 0,Y 453.569,Z 306.484,A -85,B 0,C 180,E1 -8443.88,E2 -8443.88} C_VEL
LIN {X 0,Y 453.564,Z 306.483,A -85,B 0,C 180,E1 -8447.471,E2 -8447.471} C_VEL
LIN {X 0,Y 453.594,Z 306.473,A -85,B 0,C 180,E1 -8451.087,E2 -8451.087} C_VEL
LIN {X 0,Y 453.68,Z 306.472,A -85,B 0,C 180,E1 -8453.775,E2 -8453.775} C_VEL
LIN {X 0,Y 453.767,Z 306.456,A -85,B 0,C 180,E1 -8457.337,E2 -8457.337} C_VEL
LIN {X 0,Y 453.826,Z 306.449,A -85,B 0,C 180,E1 -8460,E2 -8460} C_VEL
LIN {X 0,Y 453.766,Z 306.464,A -85,B 0,C 180,E1 -8462.663,E2 -8462.663} C_VEL
LIN {X 0,Y 453.682,Z 306.467,A -85,B 0,C 180,E1 -8466.225,E2 -8466.225} C_VEL
LIN {X 0,Y 453.594,Z 306.481,A -85,B 0,C 180,E1 -8468.914,E2 -8468.914} C_VEL
LIN {X 0,Y 453.565,Z 306.479,A -85,B 0,C 180,E1 -8472.529,E2 -8472.529} C_VEL
LIN {X 0,Y 453.546,Z 306.487,A -85,B 0,C 180,E1 -8476.196,E2 -8476.196} C_VEL
LIN {X 0,Y 453.522,Z 306.486,A -85,B 0,C 180,E1 -8479.041,E2 -8479.041} C_VEL
LIN {X 0,Y 453.478,Z 306.498,A -85,B 0,C 180,E1 -8481.836,E2 -8481.836} C_VEL
LIN {X 0,Y 453.5,Z 306.495,A -85,B 0,C 180,E1 -8484.735,E2 -8484.735} C_VEL
LIN {X 0,Y 453.519,Z 306.483,A -85,B 0,C 180,E1 -8487.956,E2 -8487.956} C_VEL
LIN {X 0,Y 453.466,Z 306.495,A -85,B 0,C 180,E1 -8491.525,E2 -8491.525} C_VEL
LIN {X 0,Y 453.483,Z 306.495,A -85,B 0,C 180,E1 -8494.776,E2 -8494.776} C_VEL
LIN {X 0,Y 453.465,Z 306.495,A -85,B 0,C 180,E1 -8498.312,E2 -8498.312} C_VEL
LIN {X 0,Y 453.495,Z 306.496,A -85,B 0,C 180,E1 -8500.609,E2 -8500.609} C_VEL
LIN {X 0,Y 453.532,Z 306.615,A -85,B 0,C 180,E1 -8503.13,E2 -8503.13} C_VEL
LIN {X 0,Y 455.07,Z 315.125,A -85,B 0,C 180,E1 -8504.917,E2 -8504.917} C_VEL
LIN {X 0,Y 454.643,Z 330.696,A -85,B 0,C 180,E1 -8507.902,E2 -8507.902} C_VEL
LIN {X 0,Y 454.584,Z 333.84,A -85,B 0,C 180,E1 -8508.445,E2 -8508.445} C_VEL
LIN {X 0,Y 456.247,Z 342.942,A -85,B 0,C 180,E1 -8508.697,E2 -8508.697} C_VEL
LIN {X 0,Y 457.785,Z 352.141,A -85,B 0,C 180,E1 -8508.91,E2 -8508.91} C_VEL
LIN {X 0,Y 456.924,Z 440.243,A -85,B 0,C 180,E1 -8510.339,E2 -8510.339} C_VEL
LIN {X 0,Y 456.67,Z 450.436,A -85,B 0,C 180,E1 -8510.605,E2 -8510.605} C_VEL
LIN {X 0,Y 456.406,Z 460.702,A -85,B 0,C 180,E1 -8510.993,E2 -8510.993} C_VEL
LIN {X 0,Y 456.054,Z 470.084,A -85,B 0,C 180,E1 -8511.453,E2 -8511.453} C_VEL
LIN {X 0,Y 455.624,Z 479.648,A -85,B 0,C 180,E1 -8512.043,E2 -8512.043} C_VEL
LIN {X 0,Y 455.105,Z 489.834,A -85,B 0,C 180,E1 -8512.829,E2 -8512.829} C_VEL
LIN {X 0,Y 454.631,Z 498.488,A -85,B 0,C 180,E1 -8513.637,E2 -8513.637} C_VEL
LIN {X 0,Y 454.162,Z 506.503,A -85,B 0,C 180,E1 -8514.528,E2 -8514.528} C_VEL
LIN {X 0,Y 453.725,Z 514.329,A -85,B 0,C 180,E1 -8515.572,E2 -8515.572} C_VEL
LIN {X 0,Y 453.252,Z 522.203,A -85,B 0,C 180,E1 -8516.857,E2 -8516.857} C_VEL
LIN {X 0,Y 452.948,Z 528.683,A -85,B 0,C 180,E1 -8518.16,E2 -8518.16} C_VEL
LIN {X 0,Y 452.808,Z 532.977,A -85,B 0,C 180,E1 -8519.19,E2 -8519.19} C_VEL
LIN {X 0,Y 452.65,Z 536.44,A -85,B 0,C 180,E1 -8520.211,E2 -8520.211} C_VEL
LIN {X 0,Y 451.919,Z 538.53,A -85,B 0,C 180,E1 -8520.904,E2 -8520.904} C_VEL
LIN {X 0,Y 448.92,Z 541.283,A -85,B 0,C 180,E1 -8522.055,E2 -8522.055} C_VEL
LIN {X 0,Y 445.912,Z 543.377,A -85,B 0,C 180,E1 -8523.246,E2 -8523.246} C_VEL
LIN {X 0,Y 445.185,Z 544.186,A -85,B 0,C 180,E1 -8523.996,E2 -8523.996} C_VEL
LIN {X 0,Y 445.163,Z 544.866,A -85,B 0,C 180,E1 -8524.769,E2 -8524.769} C_VEL
LIN {X 0,Y 445.16,Z 545.211,A -85,B 0,C 180,E1 -8526.303,E2 -8526.303} C_VEL
LIN {X 0,Y 445.176,Z 544.526,A -85,B 0,C 180,E1 -8527.735,E2 -8527.735} C_VEL
LIN {X 0,Y 445.238,Z 543.483,A -85,B 0,C 180,E1 -8528.712,E2 -8528.712} C_VEL
LIN {X 0,Y 445.45,Z 539.955,A -85,B 0,C 180,E1 -8530.651,E2 -8530.651} C_VEL
LIN {X 0,Y 445.605,Z 536.027,A -85,B 0,C 180,E1 -8532.088,E2 -8532.088} C_VEL
LIN {X 0,Y 445.744,Z 532.829,A -85,B 0,C 180,E1 -8533.041,E2 -8533.041} C_VEL
LIN {X 0,Y 446.081,Z 525.6,A -85,B 0,C 180,E1 -8534.699,E2 -8534.699} C_VEL
LIN {X 0,Y 446.432,Z 519.213,A -85,B 0,C 180,E1 -8535.877,E2 -8535.877} C_VEL
LIN {X 0,Y 446.887,Z 511.317,A -85,B 0,C 180,E1 -8537.073,E2 -8537.073} C_VEL
LIN {X 0,Y 447.33,Z 504.179,A -85,B 0,C 180,E1 -8537.985,E2 -8537.985} C_VEL
LIN {X 0,Y 447.803,Z 495.488,A -85,B 0,C 180,E1 -8538.916,E2 -8538.916} C_VEL
LIN {X 0,Y 448.342,Z 486.316,A -85,B 0,C 180,E1 -8539.729,E2 -8539.729} C_VEL
LIN {X 0,Y 448.785,Z 476.937,A -85,B 0,C 180,E1 -8540.416,E2 -8540.416} C_VEL
LIN {X 0,Y 449.266,Z 465.837,A -85,B 0,C 180,E1 -8541.057,E2 -8541.057} C_VEL
LIN {X 0,Y 449.655,Z 454.614,A -85,B 0,C 180,E1 -8541.546,E2 -8541.546} C_VEL
LIN {X 0,Y 450.008,Z 443.231,A -85,B 0,C 180,E1 -8541.892,E2 -8541.892} C_VEL
LIN {X 0,Y 450.201,Z 424.731,A -85,B 0,C 180,E1 -8542.234,E2 -8542.234} C_VEL
LIN {X 0,Y 450.742,Z 351.723,A -85,B 0,C 180,E1 -8543.411,E2 -8543.411} C_VEL
LIN {X 0,Y 447.669,Z 334.782,A -85,B 0,C 180,E1 -8543.832,E2 -8543.832} C_VEL
LIN {X 0,Y 447.63,Z 333.953,A -85,B 0,C 180,E1 -8543.917,E2 -8543.917} C_VEL
LIN {X 0,Y 448.39,Z 318.989,A -85,B 0,C 180,E1 -8547.08,E2 -8547.08} C_VEL
LIN {X 0,Y 447.848,Z 313.971,A -85,B 0,C 180,E1 -8548.202,E2 -8548.202} C_VEL
LIN {X 0,Y 446.816,Z 307.637,A -85,B 0,C 180,E1 -8549.662,E2 -8549.662} C_VEL
LIN {X 0,Y 446.795,Z 307.333,A -85,B 0,C 180,E1 -8550,E2 -8550} C_VEL
LIN {X 0,Y 446.71,Z 307.343,A -85,B 0,C 180,E1 -8552.705,E2 -8552.705} C_VEL
LIN {X 0,Y 446.637,Z 307.344,A -85,B 0,C 180,E1 -8556.324,E2 -8556.324} C_VEL
LIN {X 0,Y 446.535,Z 307.36,A -85,B 0,C 180,E1 -8559.056,E2 -8559.056} C_VEL
LIN {X 0,Y 446.523,Z 307.357,A -85,B 0,C 180,E1 -8562.73,E2 -8562.73} C_VEL
LIN {X 0,Y 446.498,Z 307.368,A -85,B 0,C 180,E1 -8566.228,E2 -8566.228} C_VEL
LIN {X 0,Y 446.471,Z 307.362,A -85,B 0,C 180,E1 -8569.303,E2 -8569.303} C_VEL
LIN {X 0,Y 446.42,Z 307.377,A -85,B 0,C 180,E1 -8572.2,E2 -8572.2} C_VEL
LIN {X 0,Y 446.451,Z 307.372,A -85,B 0,C 180,E1 -8575.153,E2 -8575.153} C_VEL
LIN {X 0,Y 446.486,Z 307.358,A -85,B 0,C 180,E1 -8578.179,E2 -8578.179} C_VEL
LIN {X 0,Y 446.421,Z 307.373,A -85,B 0,C 180,E1 -8581.775,E2 -8581.775} C_VEL
LIN {X 0,Y 446.43,Z 307.362,A -85,B 0,C 180,E1 -8584.523,E2 -8584.523} C_VEL
LIN {X 0,Y 446.416,Z 307.378,A -85,B 0,C 180,E1 -8588.079,E2 -8588.079} C_VEL
LIN {X 0,Y 446.428,Z 307.362,A -85,B 0,C 180,E1 -8590.918,E2 -8590.918} C_VEL
LIN {X 0,Y 446.399,Z 307.372,A -85,B 0,C 180,E1 -8593.846,E2 -8593.846} C_VEL
LIN {X 0,Y 446.4,Z 307.381,A -85,B 0,C 180,E1 -8596.404,E2 -8596.404} C_VEL
LIN {X 0,Y 446.424,Z 307.364,A -85,B 0,C 180,E1 -8599.083,E2 -8599.083} C_VEL
LIN {X 0,Y 446.409,Z 307.365,A -85,B 0,C 180,E1 -8602.121,E2 -8602.121} C_VEL
LIN {X 0,Y 446.425,Z 307.378,A -85,B 0,C 180,E1 -8605.476,E2 -8605.476} C_VEL
LIN {X 0,Y 446.417,Z 307.364,A -85,B 0,C 180,E1 -8608.7,E2 -8608.7} C_VEL
LIN {X 0,Y 446.45,Z 307.358,A -85,B 0,C 180,E1 -8611.83,E2 -8611.83} C_VEL
LIN {X 0,Y 446.441,Z 307.369,A -85,B 0,C 180,E1 -8614.847,E2 -8614.847} C_VEL
LIN {X 0,Y 446.451,Z 307.372,A -85,B 0,C 180,E1 -8618.245,E2 -8618.245} C_VEL
LIN {X 0,Y 446.452,Z 307.347,A -85,B 0,C 180,E1 -8621.649,E2 -8621.649} C_VEL
LIN {X 0,Y 446.509,Z 307.353,A -85,B 0,C 180,E1 -8624.48,E2 -8624.48} C_VEL
LIN {X 0,Y 446.518,Z 307.359,A -85,B 0,C 180,E1 -8628.193,E2 -8628.193} C_VEL
LIN {X 0,Y 446.527,Z 307.354,A -85,B 0,C 180,E1 -8630.944,E2 -8630.944} C_VEL
LIN {X 0,Y 446.609,Z 307.335,A -85,B 0,C 180,E1 -8633.676,E2 -8633.676} C_VEL
LIN {X 0,Y 446.657,Z 307.338,A -85,B 0,C 180,E1 -8637.294,E2 -8637.294} C_VEL
LIN {X 0,Y 446.763,Z 307.331,A -85,B 0,C 180,E1 -8640,E2 -8640} C_VEL
LIN {X 0,Y 446.655,Z 307.338,A -85,B 0,C 180,E1 -8642.705,E2 -8642.705} C_VEL
LIN {X 0,Y 446.627,Z 307.335,A -85,B 0,C 180,E1 -8646.324,E2 -8646.324} C_VEL
LIN {X 0,Y 446.528,Z 307.362,A -85,B 0,C 180,E1 -8649.055,E2 -8649.055} C_VEL
LIN {X 0,Y 446.523,Z 307.356,A -85,B 0,C 180,E1 -8652.729,E2 -8652.729} C_VEL
LIN {X 0,Y 446.451,Z 307.366,A -85,B 0,C 180,E1 -8656.207,E2 -8656.207} C_VEL
LIN {X 0,Y 446.469,Z 307.366,A -85,B 0,C 180,E1 -8659.303,E2 -8659.303} C_VEL
LIN {X 0,Y 446.419,Z 307.375,A -85,B 0,C 180,E1 -8662.199,E2 -8662.199} C_VEL
LIN {X 0,Y 446.429,Z 307.369,A -85,B 0,C 180,E1 -8665.154,E2 -8665.154} C_VEL
LIN {X 0,Y 446.437,Z 307.37,A -85,B 0,C 180,E1 -8668.182,E2 -8668.182} C_VEL
LIN {X 0,Y 446.408,Z 307.372,A -85,B 0,C 180,E1 -8671.301,E2 -8671.301} C_VEL
LIN {X 0,Y 446.421,Z 307.372,A -85,B 0,C 180,E1 -8674.523,E2 -8674.523} C_VEL
LIN {X 0,Y 446.403,Z 307.377,A -85,B 0,C 180,E1 -8678.077,E2 -8678.077} C_VEL
LIN {X 0,Y 446.398,Z 307.375,A -85,B 0,C 180,E1 -8681.394,E2 -8681.394} C_VEL
LIN {X 0,Y 446.416,Z 307.373,A -85,B 0,C 180,E1 -8685.108,E2 -8685.108} C_VEL
LIN {X 0,Y 446.398,Z 307.382,A -85,B 0,C 180,E1 -8688.605,E2 -8688.605} C_VEL
LIN {X 0,Y 446.405,Z 307.373,A -85,B 0,C 180,E1 -8691.922,E2 -8691.922} C_VEL
LIN {X 0,Y 446.42,Z 307.374,A -85,B 0,C 180,E1 -8695.476,E2 -8695.476} C_VEL
LIN {X 0,Y 446.412,Z 307.375,A -85,B 0,C 180,E1 -8698.699,E2 -8698.699} C_VEL
LIN {X 0,Y 446.448,Z 307.374,A -85,B 0,C 180,E1 -8701.83,E2 -8701.83} C_VEL
LIN {X 0,Y 446.497,Z 307.509,A -85,B 0,C 180,E1 -8704.413,E2 -8704.413} C_VEL
LIN {X 0,Y 448.694,Z 319.154,A -85,B 0,C 180,E1 -8706.947,E2 -8706.947} C_VEL
LIN {X 0,Y 448.616,Z 323.989,A -85,B 0,C 180,E1 -8707.915,E2 -8707.915} C_VEL
LIN {X 0,Y 447.77,Z 339.653,A -85,B 0,C 180,E1 -8710.993,E2 -8710.993} C_VEL
LIN {X 0,Y 447.511,Z 345.972,A -85,B 0,C 180,E1 -8712.18,E2 -8712.18} C_VEL
LIN {X 0,Y 450.824,Z 366.336,A -85,B 0,C 180,E1 -8712.671,E2 -8712.671} C_VEL
LIN {X 0,Y 450.042,Z 452.246,A -85,B 0,C 180,E1 -8714.082,E2 -8714.082} C_VEL
LIN {X 0,Y 449.781,Z 462.005,A -85,B 0,C 180,E1 -8714.334,E2 -8714.334} C_VEL
LIN {X 0,Y 449.391,Z 471.938,A -85,B 0,C 180,E1 -8714.698,E2 -8714.698} C_VEL
LIN {X 0,Y 448.922,Z 483.191,A -85,B 0,C 180,E1 -8715.262,E2 -8715.262} C_VEL
LIN {X 0,Y 448.422,Z 493.67,A -85,B 0,C 180,E1 -8715.941,E2 -8715.941} C_VEL
LIN {X 0,Y 447.925,Z 503.259,A -85,B 0,C 180,E1 -8716.71,E2 -8716.71} C_VEL
LIN {X 0,Y 447.464,Z 511.726,A -85,B 0,C 180,E1 -8717.528,E2 -8717.528} C_VEL
LIN {X 0,Y 447.006,Z 519.646,A -85,B 0,C 180,E1 -8718.436,E2 -8718.436} C_VEL
LIN {X 0,Y 446.512,Z 527.854,A -85,B 0,C 180,E1 -8719.571,E2 -8719.571} C_VEL
LIN {X 0,Y 446.117,Z 534.69,A -85,B 0,C 180,E1 -8720.707,E2 -8720.707} C_VEL
LIN {X 0,Y 445.856,Z 540.407,A -85,B 0,C 180,E1 -8721.844,E2 -8721.844} C_VEL
LIN {X 0,Y 445.643,Z 545.946,A -85,B 0,C 180,E1 -8723.208,E2 -8723.208} C_VEL
LIN {X 0,Y 445.51,Z 550.299,A -85,B 0,C 180,E1 -8724.569,E2 -8724.569} C_VEL
LIN {X 0,Y 445.412,Z 552.612,A -85,B 0,C 180,E1 -8725.475,E2 -8725.475} C_VEL
LIN {X 0,Y 445.393,Z 555.896,A -85,B 0,C 180,E1 -8727.287,E2 -8727.287} C_VEL
LIN {X 0,Y 445.309,Z 557.442,A -85,B 0,C 180,E1 -8729.096,E2 -8729.096} C_VEL
LIN {X 0,Y 445.31,Z 557.74,A -85,B 0,C 180,E1 -8730,E2 -8730} C_VEL
LIN {X 0,Y 445.345,Z 556.884,A -85,B 0,C 180,E1 -8731.809,E2 -8731.809} C_VEL
LIN {X 0,Y 445.393,Z 555.914,A -85,B 0,C 180,E1 -8732.713,E2 -8732.713} C_VEL
LIN {X 0,Y 445.412,Z 552.666,A -85,B 0,C 180,E1 -8734.525,E2 -8734.525} C_VEL
LIN {X 0,Y 445.519,Z 548.315,A -85,B 0,C 180,E1 -8736.108,E2 -8736.108} C_VEL
LIN {X 0,Y 445.686,Z 544.338,A -85,B 0,C 180,E1 -8737.247,E2 -8737.247} C_VEL
LIN {X 0,Y 445.969,Z 538.346,A -85,B 0,C 180,E1 -8738.61,E2 -8738.61} C_VEL
LIN {X 0,Y 446.263,Z 532.284,A -85,B 0,C 180,E1 -8739.747,E2 -8739.747} C_VEL
LIN {X 0,Y 446.675,Z 524.974,A -85,B 0,C 180,E1 -8740.883,E2 -8740.883} C_VEL
LIN {X 0,Y 447.263,Z 516.083,A -85,B 0,C 180,E1 -8742.017,E2 -8742.017} C_VEL
LIN {X 0,Y 447.809,Z 506.808,A -85,B 0,C 180,E1 -8742.993,E2 -8742.993} C_VEL
LIN {X 0,Y 448.293,Z 497.123,A -85,B 0,C 180,E1 -8743.832,E2 -8743.832} C_VEL
LIN {X 0,Y 448.736,Z 487.525,A -85,B 0,C 180,E1 -8744.512,E2 -8744.512} C_VEL
LIN {X 0,Y 449.263,Z 477.574,A -85,B 0,C 180,E1 -8745.074,E2 -8745.074} C_VEL
LIN {X 0,Y 449.7,Z 466.48,A -85,B 0,C 180,E1 -8745.552,E2 -8745.552} C_VEL
LIN {X 0,Y 450.026,Z 455.42,A -85,B 0,C 180,E1 -8745.889,E2 -8745.889} C_VEL
LIN {X 0,Y 450.274,Z 438.79,A -85,B 0,C 180,E1 -8746.2,E2 -8746.2} C_VEL
LIN {X 0,Y 450.776,Z 364.988,A -85,B 0,C 180,E1 -8747.403,E2 -8747.403} C_VEL
LIN {X 0,Y 447.558,Z 345.861,A -85,B 0,C 180,E1 -8747.878,E2 -8747.878} C_VEL
LIN {X 0,Y 447.663,Z 342.065,A -85,B 0,C 180,E1 -8748.537,E2 -8748.537} C_VEL
LIN {X 0,Y 448.441,Z 326.093,A -85,B 0,C 180,E1 -8751.61,E2 -8751.61} C_VEL
LIN {X 0,Y 448.78,Z 320.553,A -85,B 0,C 180,E1 -8752.686,E2 -8752.686} C_VEL
LIN {X 0,Y 447.473,Z 312.489,A -85,B 0,C 180,E1 -8754.364,E2 -8754.364} C_VEL
LIN {X 0,Y 446.453,Z 307.465,A -85,B 0,C 180,E1 -8755.496,E2 -8755.496} C_VEL
LIN {X 0,Y 446.438,Z 307.376,A -85,B 0,C 180,E1 -8758.182,E2 -8758.182} C_VEL
LIN {X 0,Y 446.412,Z 307.375,A -85,B 0,C 180,E1 -8761.301,E2 -8761.301} C_VEL
LIN {X 0,Y 446.421,Z 307.377,A -85,B 0,C 180,E1 -8764.524,E2 -8764.524} C_VEL
LIN {X 0,Y 446.412,Z 307.374,A -85,B 0,C 180,E1 -8768.079,E2 -8768.079} C_VEL
LIN {X 0,Y 446.42,Z 307.373,A -85,B 0,C 180,E1 -8770.917,E2 -8770.917} C_VEL
LIN {X 0,Y 446.399,Z 307.377,A -85,B 0,C 180,E1 -8773.846,E2 -8773.846} C_VEL
LIN {X 0,Y 446.398,Z 307.375,A -85,B 0,C 180,E1 -8776.404,E2 -8776.404} C_VEL
LIN {X 0,Y 446.425,Z 307.371,A -85,B 0,C 180,E1 -8779.083,E2 -8779.083} C_VEL
LIN {X 0,Y 446.407,Z 307.379,A -85,B 0,C 180,E1 -8782.121,E2 -8782.121} C_VEL
LIN {X 0,Y 446.429,Z 307.369,A -85,B 0,C 180,E1 -8785.477,E2 -8785.477} C_VEL
LIN {X 0,Y 446.416,Z 307.374,A -85,B 0,C 180,E1 -8788.7,E2 -8788.7} C_VEL
LIN {X 0,Y 446.484,Z 307.364,A -85,B 0,C 180,E1 -8791.822,E2 -8791.822} C_VEL
LIN {X 0,Y 446.457,Z 307.374,A -85,B 0,C 180,E1 -8794.848,E2 -8794.848} C_VEL
LIN {X 0,Y 446.448,Z 307.367,A -85,B 0,C 180,E1 -8798.245,E2 -8798.245} C_VEL
LIN {X 0,Y 446.459,Z 307.367,A -85,B 0,C 180,E1 -8801.65,E2 -8801.65} C_VEL
LIN {X 0,Y 446.51,Z 307.36,A -85,B 0,C 180,E1 -8804.48,E2 -8804.48} C_VEL
LIN {X 0,Y 446.519,Z 307.362,A -85,B 0,C 180,E1 -8808.193,E2 -8808.193} C_VEL
LIN {X 0,Y 446.602,Z 307.35,A -85,B 0,C 180,E1 -8811.858,E2 -8811.858} C_VEL
LIN {X 0,Y 446.648,Z 307.344,A -85,B 0,C 180,E1 -8814.583,E2 -8814.583} C_VEL
LIN {X 0,Y 446.71,Z 307.335,A -85,B 0,C 180,E1 -8817.295,E2 -8817.295} C_VEL
LIN {X 0,Y 446.796,Z 307.325,A -85,B 0,C 180,E1 -8820,E2 -8820} C_VEL
LIN {X 0,Y 446.71,Z 307.344,A -85,B 0,C 180,E1 -8822.705,E2 -8822.705} C_VEL
LIN {X 0,Y 446.651,Z 307.343,A -85,B 0,C 180,E1 -8826.324,E2 -8826.324} C_VEL
LIN {X 0,Y 446.54,Z 307.36,A -85,B 0,C 180,E1 -8829.056,E2 -8829.056} C_VEL
LIN {X 0,Y 446.523,Z 307.357,A -85,B 0,C 180,E1 -8832.73,E2 -8832.73} C_VEL
LIN {X 0,Y 446.498,Z 307.364,A -85,B 0,C 180,E1 -8836.228,E2 -8836.228} C_VEL
LIN {X 0,Y 446.471,Z 307.365,A -85,B 0,C 180,E1 -8839.303,E2 -8839.303} C_VEL
LIN {X 0,Y 446.419,Z 307.378,A -85,B 0,C 180,E1 -8842.2,E2 -8842.2} C_VEL
LIN {X 0,Y 446.442,Z 307.371,A -85,B 0,C 180,E1 -8845.153,E2 -8845.153} C_VEL
LIN {X 0,Y 446.486,Z 307.36,A -85,B 0,C 180,E1 -8848.179,E2 -8848.179} C_VEL
LIN {X 0,Y 446.419,Z 307.372,A -85,B 0,C 180,E1 -8851.775,E2 -8851.775} C_VEL
LIN {X 0,Y 446.424,Z 307.371,A -85,B 0,C 180,E1 -8854.524,E2 -8854.524} C_VEL
LIN {X 0,Y 446.416,Z 307.374,A -85,B 0,C 180,E1 -8858.079,E2 -8858.079} C_VEL
LIN {X 0,Y 446.428,Z 307.378,A -85,B 0,C 180,E1 -8860.918,E2 -8860.918} C_VEL
LIN {X 0,Y 446.48,Z 307.497,A -85,B 0,C 180,E1 -8862.906,E2 -8862.906} C_VEL
LIN {X 0,Y 448.017,Z 315.294,A -85,B 0,C 180,E1 -8864.587,E2 -8864.587} C_VEL
LIN {X 0,Y 447.873,Z 325.827,A -85,B 0,C 180,E1 -8866.645,E2 -8866.645} C_VEL
LIN {X 0,Y 447.67,Z 333.835,A -85,B 0,C 180,E1 -8868.149,E2 -8868.149} C_VEL
LIN {X 0,Y 448.845,Z 340.25,A -85,B 0,C 180,E1 -8868.346,E2 -8868.346} C_VEL
LIN {X 0,Y 451.018,Z 353.132,A -85,B 0,C 180,E1 -8868.652,E2 -8868.652} C_VEL
LIN {X 0,Y 450.114,Z 440.482,A -85,B 0,C 180,E1 -8870.092,E2 -8870.092} C_VEL
LIN {X 0,Y 449.872,Z 450.286,A -85,B 0,C 180,E1 -8870.352,E2 -8870.352} C_VEL
LIN {X 0,Y 449.582,Z 460.099,A -85,B 0,C 180,E1 -8870.72,E2 -8870.72} C_VEL
LIN {X 0,Y 449.173,Z 470.742,A -85,B 0,C 180,E1 -8871.255,E2 -8871.255} C_VEL
LIN {X 0,Y 448.674,Z 481.267,A -85,B 0,C 180,E1 -8871.935,E2 -8871.935} C_VEL
LIN {X 0,Y 448.173,Z 490.485,A -85,B 0,C 180,E1 -8872.669,E2 -8872.669} C_VEL
LIN {X 0,Y 447.657,Z 499.269,A -85,B 0,C 180,E1 -8873.515,E2 -8873.515} C_VEL
LIN {X 0,Y 447.15,Z 507.335,A -85,B 0,C 180,E1 -8874.441,E2 -8874.441} C_VEL
LIN {X 0,Y 446.678,Z 515.029,A -85,B 0,C 180,E1 -8875.499,E2 -8875.499} C_VEL
LIN {X 0,Y 446.19,Z 522.95,A -85,B 0,C 180,E1 -8876.834,E2 -8876.834} C_VEL
LIN {X 0,Y 445.926,Z 528.709,A -85,B 0,C 180,E1 -8878.014,E2 -8878.014} C_VEL
LIN {X 0,Y 445.727,Z 533.397,A -85,B 0,C 180,E1 -8879.173,E2 -8879.173} C_VEL
LIN {X 0,Y 445.537,Z 538.245,A -85,B 0,C 180,E1 -8880.725,E2 -8880.725} C_VEL
LIN {X 0,Y 445.384,Z 541.413,A -85,B 0,C 180,E1 -8882.087,E2 -8882.087} C_VEL
LIN {X 0,Y 445.204,Z 543.945,A -85,B 0,C 180,E1 -8883.768,E2 -8883.768} C_VEL
LIN {X 0,Y 445.185,Z 544.186,A -85,B 0,C 180,E1 -8883.996,E2 -8883.996} C_VEL
LIN {X 0,Y 444.477,Z 544.882,A -85,B 0,C 180,E1 -8884.746,E2 -8884.746} C_VEL
LIN {X 0,Y 441.577,Z 545.328,A -85,B 0,C 180,E1 -8885.972,E2 -8885.972} C_VEL
LIN {X 0,Y 439.161,Z 545.09,A -85,B 0,C 180,E1 -8886.961,E2 -8886.961} C_VEL
LIN {X 0,Y 438.148,Z 544.659,A -85,B 0,C 180,E1 -8887.724,E2 -8887.724} C_VEL
LIN {X 0,Y 438.077,Z 544.35,A -85,B 0,C 180,E1 -8887.981,E2 -8887.981} C_VEL
LIN {X 0,Y 438.199,Z 542.708,A -85,B 0,C 180,E1 -8889.339,E2 -8889.339} C_VEL
LIN {X 0,Y 438.317,Z 540.972,A -85,B 0,C 180,E1 -8890.323,E2 -8890.323} C_VEL
LIN {X 0,Y 438.477,Z 537.372,A -85,B 0,C 180,E1 -8891.787,E2 -8891.787} C_VEL
LIN {X 0,Y 438.699,Z 532.588,A -85,B 0,C 180,E1 -8893.24,E2 -8893.24} C_VEL
LIN {X 0,Y 439.002,Z 526.454,A -85,B 0,C 180,E1 -8894.684,E2 -8894.684} C_VEL
LIN {X 0,Y 439.355,Z 520.221,A -85,B 0,C 180,E1 -8895.881,E2 -8895.881} C_VEL
LIN {X 0,Y 439.823,Z 512.536,A -85,B 0,C 180,E1 -8897.092,E2 -8897.092} C_VEL
LIN {X 0,Y 440.398,Z 503.468,A -85,B 0,C 180,E1 -8898.26,E2 -8898.26} C_VEL
LIN {X 0,Y 440.913,Z 494.603,A -85,B 0,C 180,E1 -8899.205,E2 -8899.205} C_VEL
LIN {X 0,Y 441.507,Z 485.4,A -85,B 0,C 180,E1 -8900.015,E2 -8900.015} C_VEL
LIN {X 0,Y 441.902,Z 476.831,A -85,B 0,C 180,E1 -8900.649,E2 -8900.649} C_VEL
LIN {X 0,Y 442.432,Z 465.201,A -85,B 0,C 180,E1 -8901.321,E2 -8901.321} C_VEL
LIN {X 0,Y 442.815,Z 454.544,A -85,B 0,C 180,E1 -8901.788,E2 -8901.788} C_VEL
LIN {X 0,Y 443.175,Z 443.078,A -85,B 0,C 180,E1 -8902.139,E2 -8902.139} C_VEL
LIN {X 0,Y 443.385,Z 424.467,A -85,B 0,C 180,E1 -8902.486,E2 -8902.486} C_VEL
LIN {X 0,Y 443.966,Z 352.613,A -85,B 0,C 180,E1 -8903.667,E2 -8903.667} C_VEL
LIN {X 0,Y 440.763,Z 334.976,A -85,B 0,C 180,E1 -8904.108,E2 -8904.108} C_VEL
LIN {X 0,Y 440.704,Z 334.229,A -85,B 0,C 180,E1 -8904.165,E2 -8904.165} C_VEL
LIN {X 0,Y 441.432,Z 319.787,A -85,B 0,C 180,E1 -8907.262,E2 -8907.262} C_VEL
LIN {X 0,Y 440.626,Z 313.818,A -85,B 0,C 180,E1 -8908.629,E2 -8908.629} C_VEL
LIN {X 0,Y 439.765,Z 308.276,A -85,B 0,C 180,E1 -8909.971,E2 -8909.971} C_VEL
LIN {X 0,Y 439.656,Z 308.222,A -85,B 0,C 180,E1 -8912.749,E2 -8912.749} C_VEL
LIN {X 0,Y 439.607,Z 308.221,A -85,B 0,C 180,E1 -8916.425,E2 -8916.425} C_VEL
LIN {X 0,Y 439.498,Z 308.238,A -85,B 0,C 180,E1 -8919.202,E2 -8919.202} C_VEL
LIN {X 0,Y 439.467,Z 308.237,A -85,B 0,C 180,E1 -8922.938,E2 -8922.938} C_VEL
LIN {X 0,Y 439.449,Z 308.244,A -85,B 0,C 180,E1 -8926.349,E2 -8926.349} C_VEL
LIN {X 0,Y 439.404,Z 308.243,A -85,B 0,C 180,E1 -8929.626,E2 -8929.626} C_VEL
LIN {X 0,Y 439.367,Z 308.253,A -85,B 0,C 180,E1 -8932.575,E2 -8932.575} C_VEL
LIN {X 0,Y 439.402,Z 308.247,A -85,B 0,C 180,E1 -8935.585,E2 -8935.585} C_VEL
LIN {X 0,Y 439.419,Z 308.242,A -85,B 0,C 180,E1 -8938.673,E2 -8938.673} C_VEL
LIN {X 0,Y 439.372,Z 308.249,A -85,B 0,C 180,E1 -8942.03,E2 -8942.03} C_VEL
LIN {X 0,Y 439.395,Z 308.243,A -85,B 0,C 180,E1 -8945.34,E2 -8945.34} C_VEL
LIN {X 0,Y 439.386,Z 308.248,A -85,B 0,C 180,E1 -8948.595,E2 -8948.595} C_VEL
LIN {X 0,Y 439.39,Z 308.239,A -85,B 0,C 180,E1 -8951.257,E2 -8951.257} C_VEL
LIN {X 0,Y 439.4,Z 308.251,A -85,B 0,C 180,E1 -8954.73,E2 -8954.73} C_VEL
LIN {X 0,Y 439.386,Z 308.245,A -85,B 0,C 180,E1 -8957.794,E2 -8957.794} C_VEL
LIN {X 0,Y 439.39,Z 308.236,A -85,B 0,C 180,E1 -8960.223,E2 -8960.223} C_VEL
LIN {X 0,Y 439.375,Z 308.251,A -85,B 0,C 180,E1 -8963.713,E2 -8963.713} C_VEL
LIN {X 0,Y 439.374,Z 308.251,A -85,B 0,C 180,E1 -8967.054,E2 -8967.054} C_VEL
LIN {X 0,Y 439.378,Z 308.233,A -85,B 0,C 180,E1 -8970.274,E2 -8970.274} C_VEL
LIN {X 0,Y 439.384,Z 308.242,A -85,B 0,C 180,E1 -8973.393,E2 -8973.393} C_VEL
LIN {X 0,Y 439.386,Z 308.255,A -85,B 0,C 180,E1 -8976.429,E2 -8976.429} C_VEL
LIN {X 0,Y 439.39,Z 308.239,A -85,B 0,C 180,E1 -8979.397,E2 -8979.397} C_VEL
LIN {X 0,Y 439.406,Z 308.226,A -85,B 0,C 180,E1 -8982.308,E2 -8982.308} C_VEL
LIN {X 0,Y 439.447,Z 308.242,A -85,B 0,C 180,E1 -8985.174,E2 -8985.174} C_VEL
LIN {X 0,Y 439.485,Z 308.236,A -85,B 0,C 180,E1 -8988.001,E2 -8988.001} C_VEL
LIN {X 0,Y 439.504,Z 308.225,A -85,B 0,C 180,E1 -8991.725,E2 -8991.725} C_VEL
LIN {X 0,Y 439.601,Z 308.209,A -85,B 0,C 180,E1 -8994.495,E2 -8994.495} C_VEL
LIN {X 0,Y 439.63,Z 308.222,A -85,B 0,C 180,E1 -8998.168,E2 -8998.168} C_VEL
LIN {X 0,Y 439.711,Z 308.21,A -85,B 0,C 180,E1 -9000,E2 -9000} C_VEL
LIN {X 0,Y 439.606,Z 308.215,A -85,B 0,C 180,E1 -9002.749,E2 -9002.749} C_VEL
LIN {X 0,Y 439.598,Z 308.211,A -85,B 0,C 180,E1 -9006.425,E2 -9006.425} C_VEL
LIN {X 0,Y 439.492,Z 308.241,A -85,B 0,C 180,E1 -9009.202,E2 -9009.202} C_VEL
LIN {X 0,Y 439.466,Z 308.236,A -85,B 0,C 180,E1 -9012.937,E2 -9012.937} C_VEL
LIN {X 0,Y 439.398,Z 308.243,A -85,B 0,C 180,E1 -9016.326,E2 -9016.326} C_VEL
LIN {X 0,Y 439.403,Z 308.248,A -85,B 0,C 180,E1 -9019.626,E2 -9019.626} C_VEL
LIN {X 0,Y 439.364,Z 308.246,A -85,B 0,C 180,E1 -9022.575,E2 -9022.575} C_VEL
LIN {X 0,Y 439.37,Z 308.246,A -85,B 0,C 180,E1 -9025.587,E2 -9025.587} C_VEL
LIN {X 0,Y 439.389,Z 308.253,A -85,B 0,C 180,E1 -9028.675,E2 -9028.675} C_VEL
LIN {X 0,Y 439.365,Z 308.246,A -85,B 0,C 180,E1 -9032.029,E2 -9032.029} C_VEL
LIN {X 0,Y 439.389,Z 308.255,A -85,B 0,C 180,E1 -9035.339,E2 -9035.339} C_VEL
LIN {X 0,Y 439.356,Z 308.251,A -85,B 0,C 180,E1 -9038.597,E2 -9038.597} C_VEL
LIN {X 0,Y 439.345,Z 308.255,A -85,B 0,C 180,E1 -9042.21,E2 -9042.21} C_VEL
LIN {X 0,Y 439.37,Z 308.25,A -85,B 0,C 180,E1 -9045.266,E2 -9045.266} C_VEL
LIN {X 0,Y 439.351,Z 308.256,A -85,B 0,C 180,E1 -9049.016,E2 -9049.016} C_VEL
LIN {X 0,Y 439.341,Z 308.257,A -85,B 0,C 180,E1 -9052.564,E2 -9052.564} C_VEL
LIN {X 0,Y 439.393,Z 308.252,A -85,B 0,C 180,E1 -9054.843,E2 -9054.843} C_VEL
LIN {X 0,Y 439.367,Z 308.254,A -85,B 0,C 180,E1 -9058.139,E2 -9058.139} C_VEL
LIN {X 0,Y 439.406,Z 308.25,A -85,B 0,C 180,E1 -9061.604,E2 -9061.604} C_VEL
LIN {X 0,Y 439.431,Z 308.364,A -85,B 0,C 180,E1 -9064.176,E2 -9064.176} C_VEL
LIN {X 0,Y 441.705,Z 320.084,A -85,B 0,C 180,E1 -9066.777,E2 -9066.777} C_VEL
LIN {X 0,Y 441.796,Z 323.867,A -85,B 0,C 180,E1 -9067.555,E2 -9067.555} C_VEL
LIN {X 0,Y 440.786,Z 340.719,A -85,B 0,C 180,E1 -9070.922,E2 -9070.922} C_VEL
LIN {X 0,Y 440.526,Z 345.86,A -85,B 0,C 180,E1 -9071.895,E2 -9071.895} C_VEL
LIN {X 0,Y 443.993,Z 366.485,A -85,B 0,C 180,E1 -9072.409,E2 -9072.409} C_VEL
LIN {X 0,Y 443.209,Z 451.75,A -85,B 0,C 180,E1 -9073.83,E2 -9073.83} C_VEL
LIN {X 0,Y 442.962,Z 461.653,A -85,B 0,C 180,E1 -9074.087,E2 -9074.087} C_VEL
LIN {X 0,Y 442.54,Z 471.656,A -85,B 0,C 180,E1 -9074.455,E2 -9074.455} C_VEL
LIN {X 0,Y 442.059,Z 482.955,A -85,B 0,C 180,E1 -9075.028,E2 -9075.028} C_VEL
LIN {X 0,Y 441.506,Z 493.465,A -85,B 0,C 180,E1 -9075.716,E2 -9075.716} C_VEL
LIN {X 0,Y 441.042,Z 502.209,A -85,B 0,C 180,E1 -9076.416,E2 -9076.416} C_VEL
LIN {X 0,Y 440.49,Z 511.563,A -85,B 0,C 180,E1 -9077.327,E2 -9077.327} C_VEL
LIN {X 0,Y 440.021,Z 519.497,A -85,B 0,C 180,E1 -9078.25,E2 -9078.25} C_VEL
LIN {X 0,Y 439.477,Z 527.717,A -85,B 0,C 180,E1 -9079.403,E2 -9079.403} C_VEL
LIN {X 0,Y 439.098,Z 534.562,A -85,B 0,C 180,E1 -9080.557,E2 -9080.557} C_VEL
LIN {X 0,Y 438.8,Z 540.284,A -85,B 0,C 180,E1 -9081.712,E2 -9081.712} C_VEL
LIN {X 0,Y 438.581,Z 545.828,A -85,B 0,C 180,E1 -9083.097,E2 -9083.097} C_VEL
LIN {X 0,Y 438.426,Z 550.187,A -85,B 0,C 180,E1 -9084.481,E2 -9084.481} C_VEL
LIN {X 0,Y 438.343,Z 552.501,A -85,B 0,C 180,E1 -9085.402,E2 -9085.402} C_VEL
LIN {X 0,Y 438.288,Z 555.792,A -85,B 0,C 180,E1 -9087.243,E2 -9087.243} C_VEL
LIN {X 0,Y 438.267,Z 556.758,A -85,B 0,C 180,E1 -9088.162,E2 -9088.162} C_VEL
LIN {X 0,Y 438.223,Z 557.641,A -85,B 0,C 180,E1 -9090,E2 -9090} C_VEL
LIN {X 0,Y 438.267,Z 556.789,A -85,B 0,C 180,E1 -9091.838,E2 -9091.838} C_VEL
LIN {X 0,Y 438.288,Z 555.818,A -85,B 0,C 180,E1 -9092.757,E2 -9092.757} C_VEL
LIN {X 0,Y 438.343,Z 552.574,A -85,B 0,C 180,E1 -9094.598,E2 -9094.598} C_VEL
LIN {X 0,Y 438.42,Z 548.68,A -85,B 0,C 180,E1 -9096.069,E2 -9096.069} C_VEL
LIN {X 0,Y 438.616,Z 544.252,A -85,B 0,C 180,E1 -9097.365,E2 -9097.365} C_VEL
LIN {X 0,Y 438.911,Z 538.265,A -85,B 0,C 180,E1 -9098.75,E2 -9098.75} C_VEL
LIN {X 0,Y 439.245,Z 532.211,A -85,B 0,C 180,E1 -9099.904,E2 -9099.904} C_VEL
LIN {X 0,Y 439.683,Z 524.909,A -85,B 0,C 180,E1 -9101.058,E2 -9101.058} C_VEL
LIN {X 0,Y 440.284,Z 516.03,A -85,B 0,C 180,E1 -9102.21,E2 -9102.21} C_VEL
LIN {X 0,Y 440.842,Z 507.212,A -85,B 0,C 180,E1 -9103.159,E2 -9103.159} C_VEL
LIN {X 0,Y 441.329,Z 498.596,A -85,B 0,C 180,E1 -9103.937,E2 -9103.937} C_VEL
LIN {X 0,Y 441.87,Z 487.515,A -85,B 0,C 180,E1 -9104.743,E2 -9104.743} C_VEL
LIN {X 0,Y 442.425,Z 477.59,A -85,B 0,C 180,E1 -9105.313,E2 -9105.313} C_VEL
LIN {X 0,Y 442.879,Z 466.541,A -85,B 0,C 180,E1 -9105.798,E2 -9105.798} C_VEL
LIN {X 0,Y 443.224,Z 455.574,A -85,B 0,C 180,E1 -9106.14,E2 -9106.14} C_VEL
LIN {X 0,Y 443.466,Z 440.81,A -85,B 0,C 180,E1 -9106.426,E2 -9106.426} C_VEL
LIN {X 0,Y 444.043,Z 366.169,A -85,B 0,C 180,E1 -9107.661,E2 -9107.661} C_VEL
LIN {X 0,Y 440.603,Z 345.681,A -85,B 0,C 180,E1 -9108.18,E2 -9108.18} C_VEL
LIN {X 0,Y 440.967,Z 338.32,A -85,B 0,C 180,E1 -9109.554,E2 -9109.554} C_VEL
LIN {X 0,Y 441.819,Z 322.331,A -85,B 0,C 180,E1 -9112.691,E2 -9112.691} C_VEL
LIN {X 0,Y 441.223,Z 317.411,A -85,B 0,C 180,E1 -9113.715,E2 -9113.715} C_VEL
LIN {X 0,Y 439.432,Z 308.403,A -85,B 0,C 180,E1 -9115.703,E2 -9115.703} C_VEL
LIN {X 0,Y 439.394,Z 308.254,A -85,B 0,C 180,E1 -9118.675,E2 -9118.675} C_VEL
LIN {X 0,Y 439.366,Z 308.254,A -85,B 0,C 180,E1 -9122.03,E2 -9122.03} C_VEL
LIN {X 0,Y 439.39,Z 308.251,A -85,B 0,C 180,E1 -9125.34,E2 -9125.34} C_VEL
LIN {X 0,Y 439.375,Z 308.256,A -85,B 0,C 180,E1 -9128.596,E2 -9128.596} C_VEL
LIN {X 0,Y 439.379,Z 308.254,A -85,B 0,C 180,E1 -9131.256,E2 -9131.256} C_VEL
LIN {X 0,Y 439.399,Z 308.25,A -85,B 0,C 180,E1 -9134.73,E2 -9134.73} C_VEL
LIN {X 0,Y 439.394,Z 308.25,A -85,B 0,C 180,E1 -9137.796,E2 -9137.796} C_VEL
LIN {X 0,Y 439.393,Z 308.249,A -85,B 0,C 180,E1 -9140.224,E2 -9140.224} C_VEL
LIN {X 0,Y 439.374,Z 308.256,A -85,B 0,C 180,E1 -9143.713,E2 -9143.713} C_VEL
LIN {X 0,Y 439.372,Z 308.25,A -85,B 0,C 180,E1 -9147.054,E2 -9147.054} C_VEL
LIN {X 0,Y 439.383,Z 308.254,A -85,B 0,C 180,E1 -9150.275,E2 -9150.275} C_VEL
LIN {X 0,Y 439.43,Z 308.242,A -85,B 0,C 180,E1 -9153.397,E2 -9153.397} C_VEL
LIN {X 0,Y 439.386,Z 308.25,A -85,B 0,C 180,E1 -9156.43,E2 -9156.43} C_VEL
LIN {X 0,Y 439.39,Z 308.252,A -85,B 0,C 180,E1 -9159.397,E2 -9159.397} C_VEL
LIN {X 0,Y 439.432,Z 308.239,A -85,B 0,C 180,E1 -9162.31,E2 -9162.31} C_VEL
LIN {X 0,Y 439.451,Z 308.244,A -85,B 0,C 180,E1 -9165.174,E2 -9165.174} C_VEL
LIN {X 0,Y 439.485,Z 308.241,A -85,B 0,C 180,E1 -9168.002,E2 -9168.002} C_VEL
LIN {X 0,Y 439.549,Z 308.227,A -85,B 0,C 180,E1 -9171.727,E2 -9171.727} C_VEL
LIN {X 0,Y 439.623,Z 308.22,A -85,B 0,C 180,E1 -9174.496,E2 -9174.496} C_VEL
LIN {X 0,Y 439.637,Z 308.221,A -85,B 0,C 180,E1 -9178.168,E2 -9178.168} C_VEL
LIN {X 0,Y 439.766,Z 308.201,A -85,B 0,C 180,E1 -9180,E2 -9180} C_VEL
LIN {X 0,Y 439.657,Z 308.223,A -85,B 0,C 180,E1 -9182.749,E2 -9182.749} C_VEL
LIN {X 0,Y 439.622,Z 308.22,A -85,B 0,C 180,E1 -9186.425,E2 -9186.425} C_VEL
LIN {X 0,Y 439.502,Z 308.237,A -85,B 0,C 180,E1 -9189.202,E2 -9189.202} C_VEL
LIN {X 0,Y 439.467,Z 308.237,A -85,B 0,C 180,E1 -9192.938,E2 -9192.938} C_VEL
LIN {X 0,Y 439.449,Z 308.241,A -85,B 0,C 180,E1 -9196.349,E2 -9196.349} C_VEL
LIN {X 0,Y 439.404,Z 308.248,A -85,B 0,C 180,E1 -9199.626,E2 -9199.626} C_VEL
LIN {X 0,Y 439.365,Z 308.256,A -85,B 0,C 180,E1 -9202.576,E2 -9202.576} C_VEL
LIN {X 0,Y 439.381,Z 308.25,A -85,B 0,C 180,E1 -9205.587,E2 -9205.587} C_VEL
LIN {X 0,Y 439.415,Z 308.247,A -85,B 0,C 180,E1 -9208.674,E2 -9208.674} C_VEL
LIN {X 0,Y 439.37,Z 308.251,A -85,B 0,C 180,E1 -9212.03,E2 -9212.03} C_VEL
LIN {X 0,Y 439.393,Z 308.254,A -85,B 0,C 180,E1 -9215.34,E2 -9215.34} C_VEL
LIN {X 0,Y 439.384,Z 308.25,A -85,B 0,C 180,E1 -9218.595,E2 -9218.595} C_VEL
LIN {X 0,Y 439.389,Z 308.254,A -85,B 0,C 180,E1 -9221.257,E2 -9221.257} C_VEL
LIN {X 0,Y 439.418,Z 308.298,A -85,B 0,C 180,E1 -9222.632,E2 -9222.632} C_VEL
LIN {X 0,Y 440.055,Z 311.406,A -85,B 0,C 180,E1 -9223.373,E2 -9223.373} C_VEL
LIN {X 0,Y 441.201,Z 317.919,A -85,B 0,C 180,E1 -9224.743,E2 -9224.743} C_VEL
LIN {X 0,Y 440.745,Z 332.676,A -85,B 0,C 180,E1 -9227.647,E2 -9227.647} C_VEL
LIN {X 0,Y 440.813,Z 334.448,A -85,B 0,C 180,E1 -9227.886,E2 -9227.886} C_VEL
LIN {X 0,Y 444.282,Z 353.931,A -85,B 0,C 180,E1 -9228.384,E2 -9228.384} C_VEL
LIN {X 0,Y 443.302,Z 440.422,A -85,B 0,C 180,E1 -9229.831,E2 -9229.831} C_VEL
LIN {X 0,Y 443.059,Z 450.458,A -85,B 0,C 180,E1 -9230.101,E2 -9230.101} C_VEL
LIN {X 0,Y 442.724,Z 460.957,A -85,B 0,C 180,E1 -9230.508,E2 -9230.508} C_VEL
LIN {X 0,Y 442.353,Z 470.458,A -85,B 0,C 180,E1 -9230.991,E2 -9230.991} C_VEL
LIN {X 0,Y 441.813,Z 480.746,A -85,B 0,C 180,E1 -9231.656,E2 -9231.656} C_VEL
LIN {X 0,Y 441.252,Z 490.765,A -85,B 0,C 180,E1 -9232.467,E2 -9232.467} C_VEL
LIN {X 0,Y 440.728,Z 499.072,A -85,B 0,C 180,E1 -9233.274,E2 -9233.274} C_VEL
LIN {X 0,Y 440.208,Z 507.191,A -85,B 0,C 180,E1 -9234.216,E2 -9234.216} C_VEL
LIN {X 0,Y 439.641,Z 515.749,A -85,B 0,C 180,E1 -9235.424,E2 -9235.424} C_VEL
LIN {X 0,Y 439.181,Z 522.938,A -85,B 0,C 180,E1 -9236.658,E2 -9236.658} C_VEL
LIN {X 0,Y 438.909,Z 528.611,A -85,B 0,C 180,E1 -9237.832,E2 -9237.832} C_VEL
LIN {X 0,Y 438.653,Z 533.821,A -85,B 0,C 180,E1 -9239.156,E2 -9239.156} C_VEL
LIN {X 0,Y 438.47,Z 537.246,A -85,B 0,C 180,E1 -9240.206,E2 -9240.206} C_VEL
LIN {X 0,Y 438.316,Z 541.25,A -85,B 0,C 180,E1 -9241.87,E2 -9241.87} C_VEL
LIN {X 0,Y 438.134,Z 543.613,A -85,B 0,C 180,E1 -9243.311,E2 -9243.311} C_VEL
LIN {X 0,Y 438.069,Z 544.675,A -85,B 0,C 180,E1 -9244.332,E2 -9244.332} C_VEL
LIN {X 0,Y 438.079,Z 545.292,A -85,B 0,C 180,E1 -9246.355,E2 -9246.355} C_VEL
LIN {X 0,Y 438.075,Z 544.94,A -85,B 0,C 180,E1 -9247.354,E2 -9247.354} C_VEL
LIN {X 0,Y 438.077,Z 544.35,A -85,B 0,C 180,E1 -9247.981,E2 -9247.981} C_VEL
LIN {X 0,Y 437.456,Z 543.625,A -85,B 0,C 180,E1 -9248.741,E2 -9248.741} C_VEL
LIN {X 0,Y 434.7,Z 541.702,A -85,B 0,C 180,E1 -9249.966,E2 -9249.966} C_VEL
LIN {X 0,Y 432.391,Z 539.734,A -85,B 0,C 180,E1 -9250.942,E2 -9250.942} C_VEL
LIN {X 0,Y 431.456,Z 537.943,A -85,B 0,C 180,E1 -9251.685,E2 -9251.685} C_VEL
LIN {X 0,Y 431.41,Z 537.285,A -85,B 0,C 180,E1 -9251.935,E2 -9251.935} C_VEL
LIN {X 0,Y 431.663,Z 532.108,A -85,B 0,C 180,E1 -9253.495,E2 -9253.495} C_VEL
LIN {X 0,Y 432.004,Z 526.067,A -85,B 0,C 180,E1 -9254.913,E2 -9254.913} C_VEL
LIN {X 0,Y 432.373,Z 519.739,A -85,B 0,C 180,E1 -9256.128,E2 -9256.128} C_VEL
LIN {X 0,Y 432.789,Z 513.386,A -85,B 0,C 180,E1 -9257.159,E2 -9257.159} C_VEL
LIN {X 0,Y 433.434,Z 503.78,A -85,B 0,C 180,E1 -9258.425,E2 -9258.425} C_VEL
LIN {X 0,Y 433.959,Z 494.964,A -85,B 0,C 180,E1 -9259.384,E2 -9259.384} C_VEL
LIN {X 0,Y 434.567,Z 486.089,A -85,B 0,C 180,E1 -9260.186,E2 -9260.186} C_VEL
LIN {X 0,Y 435.097,Z 475.883,A -85,B 0,C 180,E1 -9260.939,E2 -9260.939} C_VEL
LIN {X 0,Y 435.555,Z 465.792,A -85,B 0,C 180,E1 -9261.533,E2 -9261.533} C_VEL
LIN {X 0,Y 435.992,Z 454.452,A -85,B 0,C 180,E1 -9262.037,E2 -9262.037} C_VEL
LIN {X 0,Y 436.323,Z 444.232,A -85,B 0,C 180,E1 -9262.364,E2 -9262.364} C_VEL
LIN {X 0,Y 436.574,Z 425.92,A -85,B 0,C 180,E1 -9262.717,E2 -9262.717} C_VEL
LIN {X 0,Y 437.193,Z 353.482,A -85,B 0,C 180,E1 -9263.93,E2 -9263.93} C_VEL
LIN {X 0,Y 433.766,Z 334.655,A -85,B 0,C 180,E1 -9264.421,E2 -9264.421} C_VEL
LIN {X 0,Y 434.009,Z 329.045,A -85,B 0,C 180,E1 -9265.589,E2 -9265.589} C_VEL
LIN {X 0,Y 434.469,Z 320.579,A -85,B 0,C 180,E1 -9267.45,E2 -9267.45} C_VEL
LIN {X 0,Y 432.735,Z 309.316,A -85,B 0,C 180,E1 -9270.116,E2 -9270.116} C_VEL
LIN {X 0,Y 432.606,Z 309.101,A -85,B 0,C 180,E1 -9272.794,E2 -9272.794} C_VEL
LIN {X 0,Y 432.557,Z 309.1,A -85,B 0,C 180,E1 -9276.531,E2 -9276.531} C_VEL
LIN {X 0,Y 432.442,Z 309.118,A -85,B 0,C 180,E1 -9279.353,E2 -9279.353} C_VEL
LIN {X 0,Y 432.433,Z 309.113,A -85,B 0,C 180,E1 -9282.804,E2 -9282.804} C_VEL
LIN {X 0,Y 432.415,Z 309.12,A -85,B 0,C 180,E1 -9286.479,E2 -9286.479} C_VEL
LIN {X 0,Y 432.341,Z 309.126,A -85,B 0,C 180,E1 -9289.96,E2 -9289.96} C_VEL
LIN {X 0,Y 432.321,Z 309.127,A -85,B 0,C 180,E1 -9292.964,E2 -9292.964} C_VEL
LIN {X 0,Y 432.364,Z 309.124,A -85,B 0,C 180,E1 -9296.033,E2 -9296.033} C_VEL
LIN {X 0,Y 432.345,Z 309.128,A -85,B 0,C 180,E1 -9299.187,E2 -9299.187} C_VEL
LIN {X 0,Y 432.325,Z 309.126,A -85,B 0,C 180,E1 -9302.443,E2 -9302.443} C_VEL
LIN {X 0,Y 432.345,Z 309.125,A -85,B 0,C 180,E1 -9305.632,E2 -9305.632} C_VEL
LIN {X 0,Y 432.356,Z 309.124,A -85,B 0,C 180,E1 -9309.342,E2 -9309.342} C_VEL
LIN {X 0,Y 432.335,Z 309.12,A -85,B 0,C 180,E1 -9311.797,E2 -9311.797} C_VEL
LIN {X 0,Y 432.335,Z 309.13,A -85,B 0,C 180,E1 -9314.347,E2 -9314.347} C_VEL
LIN {X 0,Y 432.318,Z 309.129,A -85,B 0,C 180,E1 -9317.016,E2 -9317.016} C_VEL
LIN {X 0,Y 432.315,Z 309.116,A -85,B 0,C 180,E1 -9319.824,E2 -9319.824} C_VEL
LIN {X 0,Y 432.308,Z 309.129,A -85,B 0,C 180,E1 -9323.022,E2 -9323.022} C_VEL
LIN {X 0,Y 432.36,Z 309.124,A -85,B 0,C 180,E1 -9325.997,E2 -9325.997} C_VEL
LIN {X 0,Y 432.348,Z 309.118,A -85,B 0,C 180,E1 -9329.49,E2 -9329.49} C_VEL
LIN {X 0,Y 432.346,Z 309.114,A -85,B 0,C 180,E1 -9331.874,E2 -9331.874} C_VEL
LIN {X 0,Y 432.38,Z 309.12,A -85,B 0,C 180,E1 -9335.539,E2 -9335.539} C_VEL
LIN {X 0,Y 432.352,Z 309.118,A -85,B 0,C 180,E1 -9339.046,E2 -9339.046} C_VEL
LIN {X 0,Y 432.362,Z 309.101,A -85,B 0,C 180,E1 -9342.01,E2 -9342.01} C_VEL
LIN {X 0,Y 432.395,Z 309.116,A -85,B 0,C 180,E1 -9344.926,E2 -9344.926} C_VEL
LIN {X 0,Y 432.461,Z 309.112,A -85,B 0,C 180,E1 -9347.803,E2 -9347.803} C_VEL
LIN {X 0,Y 432.464,Z 309.104,A -85,B 0,C 180,E1 -9351.59,E2 -9351.59} C_VEL
LIN {X 0,Y 432.575,Z 309.085,A -85,B 0,C 180,E1 -9354.406,E2 -9354.406} C_VEL
LIN {X 0,Y 432.599,Z 309.097,A -85,B 0,C 180,E1 -9358.138,E2 -9358.138} C_VEL
LIN {X 0,Y 432.662,Z 309.088,A -85,B 0,C 180,E1 -9360,E2 -9360} C_VEL
LIN {X 0,Y 432.56,Z 309.092,A -85,B 0,C 180,E1 -9362.794,E2 -9362.794} C_VEL
LIN {X 0,Y 432.586,Z 309.082,A -85,B 0,C 180,E1 -9365.594,E2 -9365.594} C_VEL
LIN {X 0,Y 432.464,Z 309.108,A -85,B 0,C 180,E1 -9368.41,E2 -9368.41} C_VEL
LIN {X 0,Y 432.46,Z 309.108,A -85,B 0,C 180,E1 -9372.196,E2 -9372.196} C_VEL
LIN {X 0,Y 432.386,Z 309.116,A -85,B 0,C 180,E1 -9376.04,E2 -9376.04} C_VEL
LIN {X 0,Y 432.387,Z 309.121,A -85,B 0,C 180,E1 -9379.484,E2 -9379.484} C_VEL
LIN {X 0,Y 432.311,Z 309.12,A -85,B 0,C 180,E1 -9382.964,E2 -9382.964} C_VEL
LIN {X 0,Y 432.319,Z 309.125,A -85,B 0,C 180,E1 -9386.035,E2 -9386.035} C_VEL
LIN {X 0,Y 432.326,Z 309.129,A -85,B 0,C 180,E1 -9389.188,E2 -9389.188} C_VEL
LIN {X 0,Y 432.321,Z 309.124,A -85,B 0,C 180,E1 -9392.443,E2 -9392.443} C_VEL
LIN {X 0,Y 432.335,Z 309.127,A -85,B 0,C 180,E1 -9395.818,E2 -9395.818} C_VEL
LIN {X 0,Y 432.299,Z 309.132,A -85,B 0,C 180,E1 -9399.348,E2 -9399.348} C_VEL
LIN {X 0,Y 432.301,Z 309.135,A -85,B 0,C 180,E1 -9401.8,E2 -9401.8} C_VEL
LIN {X 0,Y 432.33,Z 309.135,A -85,B 0,C 180,E1 -9404.347,E2 -9404.347} C_VEL
LIN {X 0,Y 432.298,Z 309.134,A -85,B 0,C 180,E1 -9407.018,E2 -9407.018} C_VEL
LIN {X 0,Y 432.286,Z 309.133,A -85,B 0,C 180,E1 -9409.828,E2 -9409.828} C_VEL
LIN {X 0,Y 432.301,Z 309.139,A -85,B 0,C 180,E1 -9413.021,E2 -9413.021} C_VEL
LIN {X 0,Y 432.331,Z 309.124,A -85,B 0,C 180,E1 -9416.002,E2 -9416.002} C_VEL
LIN {X 0,Y 432.344,Z 309.129,A -85,B 0,C 180,E1 -9419.49,E2 -9419.49} C_VEL
LIN {X 0,Y 432.344,Z 309.13,A -85,B 0,C 180,E1 -9421.874,E2 -9421.874} C_VEL
LIN {X 0,Y 432.389,Z 309.291,A -85,B 0,C 180,E1 -9423.969,E2 -9423.969} C_VEL
LIN {X 0,Y 434.719,Z 321.314,A -85,B 0,C 180,E1 -9426.667,E2 -9426.667} C_VEL
LIN {X 0,Y 434.859,Z 324.936,A -85,B 0,C 180,E1 -9427.428,E2 -9427.428} C_VEL
LIN {X 0,Y 433.785,Z 341.784,A -85,B 0,C 180,E1 -9430.847,E2 -9430.847} C_VEL
LIN {X 0,Y 433.585,Z 345.767,A -85,B 0,C 180,E1 -9431.604,E2 -9431.604} C_VEL
LIN {X 0,Y 437.235,Z 367.914,A -85,B 0,C 180,E1 -9432.163,E2 -9432.163} C_VEL
LIN {X 0,Y 436.403,Z 451.221,A -85,B 0,C 180,E1 -9433.571,E2 -9433.571} C_VEL
LIN {X 0,Y 436.087,Z 462.105,A -85,B 0,C 180,E1 -9433.859,E2 -9433.859} C_VEL
LIN {X 0,Y 435.699,Z 471.353,A -85,B 0,C 180,E1 -9434.205,E2 -9434.205} C_VEL
LIN {X 0,Y 435.195,Z 482.698,A -85,B 0,C 180,E1 -9434.786,E2 -9434.786} C_VEL
LIN {X 0,Y 434.609,Z 493.239,A -85,B 0,C 180,E1 -9435.484,E2 -9435.484} C_VEL
LIN {X 0,Y 434.064,Z 502.889,A -85,B 0,C 180,E1 -9436.279,E2 -9436.279} C_VEL
LIN {X 0,Y 433.527,Z 511.377,A -85,B 0,C 180,E1 -9437.12,E2 -9437.12} C_VEL
LIN {X 0,Y 433.038,Z 519.327,A -85,B 0,C 180,E1 -9438.058,E2 -9438.058} C_VEL
LIN {X 0,Y 432.47,Z 527.56,A -85,B 0,C 180,E1 -9439.229,E2 -9439.229} C_VEL
LIN {X 0,Y 432.077,Z 534.417,A -85,B 0,C 180,E1 -9440.403,E2 -9440.403} C_VEL
LIN {X 0,Y 431.759,Z 540.15,A -85,B 0,C 180,E1 -9441.576,E2 -9441.576} C_VEL
LIN {X 0,Y 431.513,Z 545.703,A -85,B 0,C 180,E1 -9442.984,E2 -9442.984} C_VEL
LIN {X 0,Y 431.327,Z 550.069,A -85,B 0,C 180,E1 -9444.389,E2 -9444.389} C_VEL
LIN {X 0,Y 431.273,Z 552.384,A -85,B 0,C 180,E1 -9445.326,E2 -9445.326} C_VEL
LIN {X 0,Y 431.185,Z 555.686,A -85,B 0,C 180,E1 -9447.197,E2 -9447.197} C_VEL
LIN {X 0,Y 431.19,Z 556.653,A -85,B 0,C 180,E1 -9448.132,E2 -9448.132} C_VEL
LIN {X 0,Y 431.138,Z 557.541,A -85,B 0,C 180,E1 -9450,E2 -9450} C_VEL
LIN {X 0,Y 431.19,Z 556.695,A -85,B 0,C 180,E1 -9451.868,E2 -9451.868} C_VEL
LIN {X 0,Y 431.184,Z 555.724,A -85,B 0,C 180,E1 -9452.803,E2 -9452.803} C_VEL
LIN {X 0,Y 431.276,Z 552.49,A -85,B 0,C 180,E1 -9454.674,E2 -9454.674} C_VEL
LIN {X 0,Y 431.366,Z 547.954,A -85,B 0,C 180,E1 -9456.368,E2 -9456.368} C_VEL
LIN {X 0,Y 431.546,Z 544.177,A -85,B 0,C 180,E1 -9457.486,E2 -9457.486} C_VEL
LIN {X 0,Y 431.877,Z 538.195,A -85,B 0,C 180,E1 -9458.893,E2 -9458.893} C_VEL
LIN {X 0,Y 432.239,Z 532.146,A -85,B 0,C 180,E1 -9460.066,E2 -9460.066} C_VEL
LIN {X 0,Y 432.702,Z 524.851,A -85,B 0,C 180,E1 -9461.239,E2 -9461.239} C_VEL
LIN {X 0,Y 433.33,Z 515.98,A -85,B 0,C 180,E1 -9462.409,E2 -9462.409} C_VEL
LIN {X 0,Y 433.868,Z 508.024,A -85,B 0,C 180,E1 -9463.292,E2 -9463.292} C_VEL
LIN {X 0,Y 434.422,Z 498.567,A -85,B 0,C 180,E1 -9464.163,E2 -9464.163} C_VEL
LIN {X 0,Y 435.011,Z 487.504,A -85,B 0,C 180,E1 -9464.981,E2 -9464.981} C_VEL
LIN {X 0,Y 435.599,Z 477.606,A -85,B 0,C 180,E1 -9465.559,E2 -9465.559} C_VEL
LIN {X 0,Y 436.062,Z 466.602,A -85,B 0,C 180,E1 -9466.052,E2 -9466.052} C_VEL
LIN {X 0,Y 436.428,Z 455.729,A -85,B 0,C 180,E1 -9466.398,E2 -9466.398} C_VEL
LIN {X 0,Y 436.691,Z 439.302,A -85,B 0,C 180,E1 -9466.719,E2 -9466.719} C_VEL
LIN {X 0,Y 437.343,Z 367.342,A -85,B 0,C 180,E1 -9467.928,E2 -9467.928} C_VEL
LIN {X 0,Y 433.686,Z 345.537,A -85,B 0,C 180,E1 -9468.497,E2 -9468.497} C_VEL
LIN {X 0,Y 434.055,Z 338.263,A -85,B 0,C 180,E1 -9469.878,E2 -9469.878} C_VEL
LIN {X 0,Y 434.849,Z 322.395,A -85,B 0,C 180,E1 -9473.049,E2 -9473.049} C_VEL
LIN {X 0,Y 432.783,Z 311.168,A -85,B 0,C 180,E1 -9475.489,E2 -9475.489} C_VEL
LIN {X 0,Y 432.371,Z 309.154,A -85,B 0,C 180,E1 -9476.032,E2 -9476.032} C_VEL
LIN {X 0,Y 432.329,Z 309.132,A -85,B 0,C 180,E1 -9479.188,E2 -9479.188} C_VEL
LIN {X 0,Y 432.32,Z 309.135,A -85,B 0,C 180,E1 -9482.443,E2 -9482.443} C_VEL
LIN {X 0,Y 432.341,Z 309.128,A -85,B 0,C 180,E1 -9485.632,E2 -9485.632} C_VEL
LIN {X 0,Y 432.337,Z 309.134,A -85,B 0,C 180,E1 -9488.714,E2 -9488.714} C_VEL
LIN {X 0,Y 432.322,Z 309.13,A -85,B 0,C 180,E1 -9491.798,E2 -9491.798} C_VEL
LIN {X 0,Y 432.332,Z 309.128,A -85,B 0,C 180,E1 -9494.348,E2 -9494.348} C_VEL
LIN {X 0,Y 432.319,Z 309.132,A -85,B 0,C 180,E1 -9497.016,E2 -9497.016} C_VEL
LIN {X 0,Y 432.332,Z 309.134,A -85,B 0,C 180,E1 -9499.821,E2 -9499.821} C_VEL
LIN {X 0,Y 432.306,Z 309.131,A -85,B 0,C 180,E1 -9503.022,E2 -9503.022} C_VEL
LIN {X 0,Y 432.359,Z 309.128,A -85,B 0,C 180,E1 -9505.997,E2 -9505.997} C_VEL
LIN {X 0,Y 432.347,Z 309.124,A -85,B 0,C 180,E1 -9509.49,E2 -9509.49} C_VEL
LIN {X 0,Y 432.392,Z 309.122,A -85,B 0,C 180,E1 -9512.929,E2 -9512.929} C_VEL
LIN {X 0,Y 432.371,Z 309.121,A -85,B 0,C 180,E1 -9516.024,E2 -9516.024} C_VEL
LIN {X 0,Y 432.351,Z 309.132,A -85,B 0,C 180,E1 -9519.046,E2 -9519.046} C_VEL
LIN {X 0,Y 432.379,Z 309.118,A -85,B 0,C 180,E1 -9522.012,E2 -9522.012} C_VEL
LIN {X 0,Y 432.398,Z 309.121,A -85,B 0,C 180,E1 -9524.927,E2 -9524.927} C_VEL
LIN {X 0,Y 432.46,Z 309.117,A -85,B 0,C 180,E1 -9527.804,E2 -9527.804} C_VEL
LIN {X 0,Y 432.493,Z 309.104,A -85,B 0,C 180,E1 -9531.591,E2 -9531.591} C_VEL
LIN {X 0,Y 432.6,Z 309.096,A -85,B 0,C 180,E1 -9534.406,E2 -9534.406} C_VEL
LIN {X 0,Y 432.607,Z 309.097,A -85,B 0,C 180,E1 -9538.138,E2 -9538.138} C_VEL
LIN {X 0,Y 432.736,Z 309.076,A -85,B 0,C 180,E1 -9540,E2 -9540} C_VEL
LIN {X 0,Y 432.606,Z 309.101,A -85,B 0,C 180,E1 -9542.794,E2 -9542.794} C_VEL
LIN {X 0,Y 432.576,Z 309.098,A -85,B 0,C 180,E1 -9546.53,E2 -9546.53} C_VEL
LIN {X 0,Y 432.445,Z 309.117,A -85,B 0,C 180,E1 -9549.353,E2 -9549.353} C_VEL
LIN {X 0,Y 432.432,Z 309.112,A -85,B 0,C 180,E1 -9552.804,E2 -9552.804} C_VEL
LIN {X 0,Y 432.414,Z 309.117,A -85,B 0,C 180,E1 -9556.479,E2 -9556.479} C_VEL
LIN {X 0,Y 432.341,Z 309.131,A -85,B 0,C 180,E1 -9559.961,E2 -9559.961} C_VEL
LIN {X 0,Y 432.319,Z 309.131,A -85,B 0,C 180,E1 -9562.964,E2 -9562.964} C_VEL
LIN {X 0,Y 432.34,Z 309.129,A -85,B 0,C 180,E1 -9565.002,E2 -9565.002} C_VEL
LIN {X 0,Y 432.37,Z 309.118,A -85,B 0,C 180,E1 -9568.124,E2 -9568.124} C_VEL
LIN {X 0,Y 432.321,Z 309.129,A -85,B 0,C 180,E1 -9571.346,E2 -9571.346} C_VEL
LIN {X 0,Y 432.338,Z 309.127,A -85,B 0,C 180,E1 -9574.677,E2 -9574.677} C_VEL
LIN {X 0,Y 432.339,Z 309.128,A -85,B 0,C 180,E1 -9578.15,E2 -9578.15} C_VEL
LIN {X 0,Y 432.334,Z 309.134,A -85,B 0,C 180,E1 -9581.602,E2 -9581.602} C_VEL
LIN {X 0,Y 432.384,Z 309.235,A -85,B 0,C 180,E1 -9582.419,E2 -9582.419} C_VEL
LIN {X 0,Y 434.281,Z 319.075,A -85,B 0,C 180,E1 -9584.598,E2 -9584.598} C_VEL
LIN {X 0,Y 433.831,Z 333.883,A -85,B 0,C 180,E1 -9587.523,E2 -9587.523} C_VEL
LIN {X 0,Y 434.437,Z 337.288,A -85,B 0,C 180,E1 -9587.655,E2 -9587.655} C_VEL
LIN {X 0,Y 437.546,Z 354.613,A -85,B 0,C 180,E1 -9588.103,E2 -9588.103} C_VEL
LIN {X 0,Y 436.515,Z 440.356,A -85,B 0,C 180,E1 -9589.562,E2 -9589.562} C_VEL
LIN {X 0,Y 436.253,Z 449.845,A -85,B 0,C 180,E1 -9589.814,E2 -9589.814} C_VEL
LIN {X 0,Y 435.916,Z 460.975,A -85,B 0,C 180,E1 -9590.249,E2 -9590.249} C_VEL
LIN {X 0,Y 435.489,Z 471.019,A -85,B 0,C 180,E1 -9590.772,E2 -9590.772} C_VEL
LIN {X 0,Y 434.978,Z 480.433,A -85,B 0,C 180,E1 -9591.386,E2 -9591.386} C_VEL
LIN {X 0,Y 434.413,Z 490.407,A -85,B 0,C 180,E1 -9592.198,E2 -9592.198} C_VEL
LIN {X 0,Y 433.745,Z 500.08,A -85,B 0,C 180,E1 -9593.165,E2 -9593.165} C_VEL
LIN {X 0,Y 433.281,Z 507.065,A -85,B 0,C 180,E1 -9593.986,E2 -9593.986} C_VEL
LIN {X 0,Y 432.756,Z 514.838,A -85,B 0,C 180,E1 -9595.078,E2 -9595.078} C_VEL
LIN {X 0,Y 432.205,Z 522.729,A -85,B 0,C 180,E1 -9596.436,E2 -9596.436} C_VEL
LIN {X 0,Y 431.844,Z 529.19,A -85,B 0,C 180,E1 -9597.808,E2 -9597.808} C_VEL
LIN {X 0,Y 431.577,Z 534.252,A -85,B 0,C 180,E1 -9599.139,E2 -9599.139} C_VEL
LIN {X 0,Y 431.402,Z 537.64,A -85,B 0,C 180,E1 -9600.211,E2 -9600.211} C_VEL
LIN {X 0,Y 431.237,Z 541.353,A -85,B 0,C 180,E1 -9601.795,E2 -9601.795} C_VEL
LIN {X 0,Y 431.082,Z 543.156,A -85,B 0,C 180,E1 -9602.839,E2 -9602.839} C_VEL
LIN {X 0,Y 431.026,Z 544.348,A -85,B 0,C 180,E1 -9603.881,E2 -9603.881} C_VEL
LIN {X 0,Y 430.961,Z 545.132,A -85,B 0,C 180,E1 -9604.913,E2 -9604.913} C_VEL
LIN {X 0,Y 430.977,Z 545.475,A -85,B 0,C 180,E1 -9605.952,E2 -9605.952} C_VEL
LIN {X 0,Y 430.982,Z 544.499,A -85,B 0,C 180,E1 -9607.997,E2 -9607.997} C_VEL
LIN {X 0,Y 431.088,Z 543.466,A -85,B 0,C 180,E1 -9608.982,E2 -9608.982} C_VEL
LIN {X 0,Y 431.297,Z 539.808,A -85,B 0,C 180,E1 -9610.929,E2 -9610.929} C_VEL
LIN {X 0,Y 431.41,Z 537.285,A -85,B 0,C 180,E1 -9611.935,E2 -9611.935} C_VEL
LIN {X 0,Y 430.861,Z 535.224,A -85,B 0,C 180,E1 -9612.666,E2 -9612.666} C_VEL
LIN {X 0,Y 428.217,Z 531.23,A -85,B 0,C 180,E1 -9613.823,E2 -9613.823} C_VEL
LIN {X 0,Y 425.597,Z 526.6,A -85,B 0,C 180,E1 -9614.949,E2 -9614.949} C_VEL
LIN {X 0,Y 425.107,Z 523.362,A -85,B 0,C 180,E1 -9615.621,E2 -9615.621} C_VEL
LIN {X 0,Y 425.529,Z 517.777,A -85,B 0,C 180,E1 -9616.631,E2 -9616.631} C_VEL
LIN {X 0,Y 425.93,Z 511.481,A -85,B 0,C 180,E1 -9617.614,E2 -9617.614} C_VEL
LIN {X 0,Y 426.462,Z 504.096,A -85,B 0,C 180,E1 -9618.594,E2 -9618.594} C_VEL
LIN {X 0,Y 427.013,Z 495.323,A -85,B 0,C 180,E1 -9619.57,E2 -9619.57} C_VEL
LIN {X 0,Y 427.667,Z 486.268,A -85,B 0,C 180,E1 -9620.402,E2 -9620.402} C_VEL
LIN {X 0,Y 428.198,Z 476.371,A -85,B 0,C 180,E1 -9621.149,E2 -9621.149} C_VEL
LIN {X 0,Y 428.69,Z 466.375,A -85,B 0,C 180,E1 -9621.753,E2 -9621.753} C_VEL
LIN {X 0,Y 429.155,Z 454.393,A -85,B 0,C 180,E1 -9622.295,E2 -9622.295} C_VEL
LIN {X 0,Y 429.516,Z 444.047,A -85,B 0,C 180,E1 -9622.626,E2 -9622.626} C_VEL
LIN {X 0,Y 429.742,Z 427.466,A -85,B 0,C 180,E1 -9622.955,E2 -9622.955} C_VEL
LIN {X 0,Y 430.418,Z 354.219,A -85,B 0,C 180,E1 -9624.202,E2 -9624.202} C_VEL
LIN {X 0,Y 426.84,Z 334.875,A -85,B 0,C 180,E1 -9624.716,E2 -9624.716} C_VEL
LIN {X 0,Y 426.94,Z 331.963,A -85,B 0,C 180,E1 -9625.279,E2 -9625.279} C_VEL
LIN {X 0,Y 427.501,Z 321.374,A -85,B 0,C 180,E1 -9627.645,E2 -9627.645} C_VEL
LIN {X 0,Y 425.675,Z 310.156,A -85,B 0,C 180,E1 -9630.355,E2 -9630.355} C_VEL
LIN {X 0,Y 425.557,Z 309.979,A -85,B 0,C 180,E1 -9632.84,E2 -9632.84} C_VEL
LIN {X 0,Y 425.549,Z 309.972,A -85,B 0,C 180,E1 -9635.687,E2 -9635.687} C_VEL
LIN {X 0,Y 425.41,Z 309.988,A -85,B 0,C 180,E1 -9638.551,E2 -9638.551} C_VEL
LIN {X 0,Y 425.414,Z 309.987,A -85,B 0,C 180,E1 -9642.402,E2 -9642.402} C_VEL
LIN {X 0,Y 425.39,Z 309.996,A -85,B 0,C 180,E1 -9646.312,E2 -9646.312} C_VEL
LIN {X 0,Y 425.33,Z 309.997,A -85,B 0,C 180,E1 -9649.636,E2 -9649.636} C_VEL
LIN {X 0,Y 425.29,Z 310.009,A -85,B 0,C 180,E1 -9652.339,E2 -9652.339} C_VEL
LIN {X 0,Y 425.294,Z 310.005,A -85,B 0,C 180,E1 -9655.446,E2 -9655.446} C_VEL
LIN {X 0,Y 425.333,Z 309.996,A -85,B 0,C 180,E1 -9658.632,E2 -9658.632} C_VEL
LIN {X 0,Y 425.267,Z 310.007,A -85,B 0,C 180,E1 -9661.927,E2 -9661.927} C_VEL
LIN {X 0,Y 425.3,Z 309.998,A -85,B 0,C 180,E1 -9665.336,E2 -9665.336} C_VEL
LIN {X 0,Y 425.302,Z 310.002,A -85,B 0,C 180,E1 -9669.044,E2 -9669.044} C_VEL
LIN {X 0,Y 425.276,Z 310.004,A -85,B 0,C 180,E1 -9672.653,E2 -9672.653} C_VEL
LIN {X 0,Y 425.262,Z 310.01,A -85,B 0,C 180,E1 -9676.044,E2 -9676.044} C_VEL
LIN {X 0,Y 425.267,Z 310.006,A -85,B 0,C 180,E1 -9678.62,E2 -9678.62} C_VEL
LIN {X 0,Y 425.294,Z 309.995,A -85,B 0,C 180,E1 -9681.101,E2 -9681.101} C_VEL
LIN {X 0,Y 425.3,Z 310.002,A -85,B 0,C 180,E1 -9684.664,E2 -9684.664} C_VEL
LIN {X 0,Y 425.266,Z 310.001,A -85,B 0,C 180,E1 -9688.073,E2 -9688.073} C_VEL
LIN {X 0,Y 425.312,Z 309.983,A -85,B 0,C 180,E1 -9691.366,E2 -9691.366} C_VEL
LIN {X 0,Y 425.274,Z 310.009,A -85,B 0,C 180,E1 -9694.553,E2 -9694.553} C_VEL
LIN {X 0,Y 425.306,Z 310.005,A -85,B 0,C 180,E1 -9696.635,E2 -9696.635} C_VEL
LIN {X 0,Y 425.33,Z 309.993,A -85,B 0,C 180,E1 -9700.365,E2 -9700.365} C_VEL
LIN {X 0,Y 425.39,Z 309.982,A -85,B 0,C 180,E1 -9703.688,E2 -9703.688} C_VEL
LIN {X 0,Y 425.414,Z 309.992,A -85,B 0,C 180,E1 -9707.598,E2 -9707.598} C_VEL
LIN {X 0,Y 425.408,Z 309.985,A -85,B 0,C 180,E1 -9711.449,E2 -9711.449} C_VEL
LIN {X 0,Y 425.529,Z 309.962,A -85,B 0,C 180,E1 -9714.313,E2 -9714.313} C_VEL
LIN {X 0,Y 425.568,Z 309.972,A -85,B 0,C 180,E1 -9718.107,E2 -9718.107} C_VEL
LIN {X 0,Y 425.511,Z 309.975,A -85,B 0,C 180,E1 -9720.946,E2 -9720.946} C_VEL
LIN {X 0,Y 425.515,Z 309.968,A -85,B 0,C 180,E1 -9722.84,E2 -9722.84} C_VEL
LIN {X 0,Y 425.542,Z 309.959,A -85,B 0,C 180,E1 -9725.687,E2 -9725.687} C_VEL
LIN {X 0,Y 425.408,Z 309.987,A -85,B 0,C 180,E1 -9728.55,E2 -9728.55} C_VEL
LIN {X 0,Y 425.413,Z 309.985,A -85,B 0,C 180,E1 -9732.401,E2 -9732.401} C_VEL
LIN {X 0,Y 425.3,Z 309.99,A -85,B 0,C 180,E1 -9735.331,E2 -9735.331} C_VEL
